// ---- DUTs/IO/PdoEntries/FSOE_BAA7477B.TcDUT
{attribute 'GeneratedUsingTerminal: EK1960-2600-0019'}
{attribute addProperty BoxType "EK1960-2600-0019"}
{attribute addProperty Id "FSoE_CommandUSINT1FSOUT_Module_1_Module_FaultBOOL1FSOUT_Module_2_Module_FaultBOOL1FSOUT_Module_3_Module_FaultBOOL1FSOUT_Module_4_Module_FaultBOOL1FSOUT_Module_5_Module_FaultBOOL1FSOUT_Module_6_Module_FaultBOOL1FSOUT_Relais_Module_Module_FaultBOOL1FSIN_Module_1_Channel_1_InputBOOL1FSIN_Module_1_Channel_2_InputBOOL1FSIN_Module_1_Module_FaultBOOL1FSIN_Module_2_Channel_1_InputBOOL1FSIN_Module_2_Channel_2_InputBOOL1FSIN_Module_2_Module_FaultBOOL1FSIN_Module_3_Channel_1_InputBOOL1FSIN_Module_3_Channel_2_InputBOOL1FSIN_Module_3_Module_FaultBOOL1FSoE_CRC_000UINT2FSIN_Module_4_Channel_1_InputBOOL1FSIN_Module_4_Channel_2_InputBOOL1FSIN_Module_4_Module_FaultBOOL1FSIN_Module_5_Channel_1_InputBOOL1FSIN_Module_5_Channel_2_InputBOOL1FSIN_Module_5_Module_FaultBOOL1FSIN_Module_6_Channel_1_InputBOOL1FSIN_Module_6_Channel_2_InputBOOL1FSIN_Module_6_Module_FaultBOOL1FSIN_Module_7_Channel_1_InputBOOL1FSIN_Module_7_Channel_2_InputBOOL1FSIN_Module_7_Module_FaultBOOL1FSIN_Module_8_Channel_1_InputBOOL1FSIN_Module_8_Channel_2_InputBOOL1FSIN_Module_8_Module_FaultBOOL1FSIN_Module_9_Channel_1_InputBOOL1FSoE_CRC_001UINT2FSIN_Module_9_Channel_2_InputBOOL1FSIN_Module_9_Module_Fault_1BOOL1FSIN_Module_9_Module_Fault_2BOOL1FSIN_Module_10_Channel_1_InputBOOL1FSIN_Module_10_Channel_2_InputBOOL1FSIN_Module_10_Module_Fault_1BOOL1FSIN_Module_10_Module_Fault_2BOOL1FSoE_CRC_002UINT2FSoE_Connection_IDUINT2"}
{attribute addProperty CRC "3131524987"}
{attribute addProperty Size "48"}
TYPE FSOE_BAA7477B :
STRUCT
	{attribute addProperty Name "FSoE_Command"}
	FSoE_Command : USINT;
	{attribute addProperty Name "FSOUT_Module_1_Module_Fault"}
	FSOUT_Module_1_Module_Fault : BOOL;
	{attribute addProperty Name "FSOUT_Module_2_Module_Fault"}
	FSOUT_Module_2_Module_Fault : BOOL;
	{attribute addProperty Name "FSOUT_Module_3_Module_Fault"}
	FSOUT_Module_3_Module_Fault : BOOL;
	{attribute addProperty Name "FSOUT_Module_4_Module_Fault"}
	FSOUT_Module_4_Module_Fault : BOOL;
	{attribute addProperty Name "FSOUT_Module_5_Module_Fault"}
	FSOUT_Module_5_Module_Fault : BOOL;
	{attribute addProperty Name "FSOUT_Module_6_Module_Fault"}
	FSOUT_Module_6_Module_Fault : BOOL;
	{attribute addProperty Name "FSOUT_Relais_Module_Module_Fault"}
	FSOUT_Relais_Module_Module_Fault : BOOL;
	{attribute addProperty Name "FSIN_Module_1_Channel_1_Input"}
	FSIN_Module_1_Channel_1_Input : BOOL;
	{attribute addProperty Name "FSIN_Module_1_Channel_2_Input"}
	FSIN_Module_1_Channel_2_Input : BOOL;
	{attribute addProperty Name "FSIN_Module_1_Module_Fault"}
	FSIN_Module_1_Module_Fault : BOOL;
	{attribute addProperty Name "FSIN_Module_2_Channel_1_Input"}
	FSIN_Module_2_Channel_1_Input : BOOL;
	{attribute addProperty Name "FSIN_Module_2_Channel_2_Input"}
	FSIN_Module_2_Channel_2_Input : BOOL;
	{attribute addProperty Name "FSIN_Module_2_Module_Fault"}
	FSIN_Module_2_Module_Fault : BOOL;
	{attribute addProperty Name "FSIN_Module_3_Channel_1_Input"}
	FSIN_Module_3_Channel_1_Input : BOOL;
	{attribute addProperty Name "FSIN_Module_3_Channel_2_Input"}
	FSIN_Module_3_Channel_2_Input : BOOL;
	{attribute addProperty Name "FSIN_Module_3_Module_Fault"}
	FSIN_Module_3_Module_Fault : BOOL;
	{attribute addProperty Name "FSoE_CRC_000"}
	FSoE_CRC_000 : UINT;
	{attribute addProperty Name "FSIN_Module_4_Channel_1_Input"}
	FSIN_Module_4_Channel_1_Input : BOOL;
	{attribute addProperty Name "FSIN_Module_4_Channel_2_Input"}
	FSIN_Module_4_Channel_2_Input : BOOL;
	{attribute addProperty Name "FSIN_Module_4_Module_Fault"}
	FSIN_Module_4_Module_Fault : BOOL;
	{attribute addProperty Name "FSIN_Module_5_Channel_1_Input"}
	FSIN_Module_5_Channel_1_Input : BOOL;
	{attribute addProperty Name "FSIN_Module_5_Channel_2_Input"}
	FSIN_Module_5_Channel_2_Input : BOOL;
	{attribute addProperty Name "FSIN_Module_5_Module_Fault"}
	FSIN_Module_5_Module_Fault : BOOL;
	{attribute addProperty Name "FSIN_Module_6_Channel_1_Input"}
	FSIN_Module_6_Channel_1_Input : BOOL;
	{attribute addProperty Name "FSIN_Module_6_Channel_2_Input"}
	FSIN_Module_6_Channel_2_Input : BOOL;
	{attribute addProperty Name "FSIN_Module_6_Module_Fault"}
	FSIN_Module_6_Module_Fault : BOOL;
	{attribute addProperty Name "FSIN_Module_7_Channel_1_Input"}
	FSIN_Module_7_Channel_1_Input : BOOL;
	{attribute addProperty Name "FSIN_Module_7_Channel_2_Input"}
	FSIN_Module_7_Channel_2_Input : BOOL;
	{attribute addProperty Name "FSIN_Module_7_Module_Fault"}
	FSIN_Module_7_Module_Fault : BOOL;
	{attribute addProperty Name "FSIN_Module_8_Channel_1_Input"}
	FSIN_Module_8_Channel_1_Input : BOOL;
	{attribute addProperty Name "FSIN_Module_8_Channel_2_Input"}
	FSIN_Module_8_Channel_2_Input : BOOL;
	{attribute addProperty Name "FSIN_Module_8_Module_Fault"}
	FSIN_Module_8_Module_Fault : BOOL;
	{attribute addProperty Name "FSIN_Module_9_Channel_1_Input"}
	FSIN_Module_9_Channel_1_Input : BOOL;
	{attribute addProperty Name "FSoE_CRC_001"}
	FSoE_CRC_001 : UINT;
	{attribute addProperty Name "FSIN_Module_9_Channel_2_Input"}
	FSIN_Module_9_Channel_2_Input : BOOL;
	{attribute addProperty Name "FSIN_Module_9_Module_Fault_1"}
	FSIN_Module_9_Module_Fault_1 : BOOL;
	{attribute addProperty Name "FSIN_Module_9_Module_Fault_2"}
	FSIN_Module_9_Module_Fault_2 : BOOL;
	{attribute addProperty Name "FSIN_Module_10_Channel_1_Input"}
	FSIN_Module_10_Channel_1_Input : BOOL;
	{attribute addProperty Name "FSIN_Module_10_Channel_2_Input"}
	FSIN_Module_10_Channel_2_Input : BOOL;
	{attribute addProperty Name "FSIN_Module_10_Module_Fault_1"}
	FSIN_Module_10_Module_Fault_1 : BOOL;
	{attribute addProperty Name "FSIN_Module_10_Module_Fault_2"}
	FSIN_Module_10_Module_Fault_2 : BOOL;
	{attribute addProperty Name "FSoE_CRC_002"}
	FSoE_CRC_002 : UINT;
	{attribute addProperty Name "FSoE_Connection_ID"}
	FSoE_Connection_ID : UINT;
END_STRUCT
END_TYPE

// ---- DUTs/IO/PdoEntries/FSOE_CEFF8C56.TcDUT
{attribute 'GeneratedUsingTerminal: EK1960-2600-0019'}
{attribute addProperty BoxType "EK1960-2600-0019"}
{attribute addProperty Id "FSoE_CommandUSINT1FSOUT_Module_1_Channel_1_OutputBOOL1FSOUT_Module_1_Channel_2_OutputBOOL1FSOUT_Module_1_Channel_3_OutputBOOL1FSOUT_Module_1_Channel_4_OutputBOOL1FSOUT_Module_1_ErrAckBOOL1FSOUT_Module_2_Channel_1_OutputBOOL1FSOUT_Module_2_Channel_2_OutputBOOL1FSOUT_Module_2_Channel_3_OutputBOOL1FSOUT_Module_2_Channel_4_OutputBOOL1FSOUT_Module_2_ErrAckBOOL1FSOUT_Module_3_Channel_1_OutputBOOL1FSOUT_Module_3_Channel_2_OutputBOOL1FSOUT_Module_3_Channel_3_OutputBOOL1FSOUT_Module_3_Channel_4_OutputBOOL1FSOUT_Module_3_ErrAckBOOL1FSOUT_Module_4_Channel_1_OutputBOOL1FSoE_CRC_000UINT2FSOUT_Module_4_Channel_2_OutputBOOL1FSOUT_Module_4_Channel_3_OutputBOOL1FSOUT_Module_4_Channel_4_OutputBOOL1FSOUT_Module_4_ErrAckBOOL1FSOUT_Module_5_Channel_1_OutputBOOL1FSOUT_Module_5_Channel_2_OutputBOOL1FSOUT_Module_5_Channel_3_OutputBOOL1FSOUT_Module_5_Channel_4_OutputBOOL1FSOUT_Module_5_ErrAckBOOL1FSOUT_Module_6_Channel_1_OutputBOOL1FSOUT_Module_6_Channel_2_OutputBOOL1FSOUT_Module_6_Channel_3_OutputBOOL1FSOUT_Module_6_Channel_4_OutputBOOL1FSOUT_Module_6_ErrAckBOOL1FSOUT_Relais_Module_Channel_1_OutputBOOL1FSOUT_Relais_Module_Channel_2_OutputBOOL1FSoE_CRC_001UINT2FSOUT_Relais_Module_Channel_3_OutputBOOL1FSOUT_Relais_Module_Channel_4_OutputBOOL1FSOUT_Relais_Module_ErrAckBOOL1FSIN_Module_1_ErrAckBOOL1FSIN_Module_2_ErrAckBOOL1FSIN_Module_3_ErrAckBOOL1FSIN_Module_4_ErrAckBOOL1FSIN_Module_5_ErrAckBOOL1FSIN_Module_6_ErrAckBOOL1FSIN_Module_7_ErrAckBOOL1FSIN_Module_8_ErrAckBOOL1FSIN_Module_9_ErrAck_1BOOL1FSIN_Module_9_ErrAck_2BOOL1FSIN_Module_10_ErrAck_1BOOL1FSIN_Module_10_ErrAck_2BOOL1FSoE_CRC_002UINT2FSoE_Connection_IDUINT2"}
{attribute addProperty CRC "3472854102"}
{attribute addProperty Size "56"}
TYPE FSOE_CEFF8C56 :
STRUCT
	{attribute addProperty Name "FSoE_Command"}
	FSoE_Command : USINT;
	{attribute addProperty Name "FSOUT_Module_1_Channel_1_Output"}
	FSOUT_Module_1_Channel_1_Output : BOOL;
	{attribute addProperty Name "FSOUT_Module_1_Channel_2_Output"}
	FSOUT_Module_1_Channel_2_Output : BOOL;
	{attribute addProperty Name "FSOUT_Module_1_Channel_3_Output"}
	FSOUT_Module_1_Channel_3_Output : BOOL;
	{attribute addProperty Name "FSOUT_Module_1_Channel_4_Output"}
	FSOUT_Module_1_Channel_4_Output : BOOL;
	{attribute addProperty Name "FSOUT_Module_1_ErrAck"}
	FSOUT_Module_1_ErrAck : BOOL;
	{attribute addProperty Name "FSOUT_Module_2_Channel_1_Output"}
	FSOUT_Module_2_Channel_1_Output : BOOL;
	{attribute addProperty Name "FSOUT_Module_2_Channel_2_Output"}
	FSOUT_Module_2_Channel_2_Output : BOOL;
	{attribute addProperty Name "FSOUT_Module_2_Channel_3_Output"}
	FSOUT_Module_2_Channel_3_Output : BOOL;
	{attribute addProperty Name "FSOUT_Module_2_Channel_4_Output"}
	FSOUT_Module_2_Channel_4_Output : BOOL;
	{attribute addProperty Name "FSOUT_Module_2_ErrAck"}
	FSOUT_Module_2_ErrAck : BOOL;
	{attribute addProperty Name "FSOUT_Module_3_Channel_1_Output"}
	FSOUT_Module_3_Channel_1_Output : BOOL;
	{attribute addProperty Name "FSOUT_Module_3_Channel_2_Output"}
	FSOUT_Module_3_Channel_2_Output : BOOL;
	{attribute addProperty Name "FSOUT_Module_3_Channel_3_Output"}
	FSOUT_Module_3_Channel_3_Output : BOOL;
	{attribute addProperty Name "FSOUT_Module_3_Channel_4_Output"}
	FSOUT_Module_3_Channel_4_Output : BOOL;
	{attribute addProperty Name "FSOUT_Module_3_ErrAck"}
	FSOUT_Module_3_ErrAck : BOOL;
	{attribute addProperty Name "FSOUT_Module_4_Channel_1_Output"}
	FSOUT_Module_4_Channel_1_Output : BOOL;
	{attribute addProperty Name "FSoE_CRC_000"}
	FSoE_CRC_000 : UINT;
	{attribute addProperty Name "FSOUT_Module_4_Channel_2_Output"}
	FSOUT_Module_4_Channel_2_Output : BOOL;
	{attribute addProperty Name "FSOUT_Module_4_Channel_3_Output"}
	FSOUT_Module_4_Channel_3_Output : BOOL;
	{attribute addProperty Name "FSOUT_Module_4_Channel_4_Output"}
	FSOUT_Module_4_Channel_4_Output : BOOL;
	{attribute addProperty Name "FSOUT_Module_4_ErrAck"}
	FSOUT_Module_4_ErrAck : BOOL;
	{attribute addProperty Name "FSOUT_Module_5_Channel_1_Output"}
	FSOUT_Module_5_Channel_1_Output : BOOL;
	{attribute addProperty Name "FSOUT_Module_5_Channel_2_Output"}
	FSOUT_Module_5_Channel_2_Output : BOOL;
	{attribute addProperty Name "FSOUT_Module_5_Channel_3_Output"}
	FSOUT_Module_5_Channel_3_Output : BOOL;
	{attribute addProperty Name "FSOUT_Module_5_Channel_4_Output"}
	FSOUT_Module_5_Channel_4_Output : BOOL;
	{attribute addProperty Name "FSOUT_Module_5_ErrAck"}
	FSOUT_Module_5_ErrAck : BOOL;
	{attribute addProperty Name "FSOUT_Module_6_Channel_1_Output"}
	FSOUT_Module_6_Channel_1_Output : BOOL;
	{attribute addProperty Name "FSOUT_Module_6_Channel_2_Output"}
	FSOUT_Module_6_Channel_2_Output : BOOL;
	{attribute addProperty Name "FSOUT_Module_6_Channel_3_Output"}
	FSOUT_Module_6_Channel_3_Output : BOOL;
	{attribute addProperty Name "FSOUT_Module_6_Channel_4_Output"}
	FSOUT_Module_6_Channel_4_Output : BOOL;
	{attribute addProperty Name "FSOUT_Module_6_ErrAck"}
	FSOUT_Module_6_ErrAck : BOOL;
	{attribute addProperty Name "FSOUT_Relais_Module_Channel_1_Output"}
	FSOUT_Relais_Module_Channel_1_Output : BOOL;
	{attribute addProperty Name "FSOUT_Relais_Module_Channel_2_Output"}
	FSOUT_Relais_Module_Channel_2_Output : BOOL;
	{attribute addProperty Name "FSoE_CRC_001"}
	FSoE_CRC_001 : UINT;
	{attribute addProperty Name "FSOUT_Relais_Module_Channel_3_Output"}
	FSOUT_Relais_Module_Channel_3_Output : BOOL;
	{attribute addProperty Name "FSOUT_Relais_Module_Channel_4_Output"}
	FSOUT_Relais_Module_Channel_4_Output : BOOL;
	{attribute addProperty Name "FSOUT_Relais_Module_ErrAck"}
	FSOUT_Relais_Module_ErrAck : BOOL;
	{attribute addProperty Name "FSIN_Module_1_ErrAck"}
	FSIN_Module_1_ErrAck : BOOL;
	{attribute addProperty Name "FSIN_Module_2_ErrAck"}
	FSIN_Module_2_ErrAck : BOOL;
	{attribute addProperty Name "FSIN_Module_3_ErrAck"}
	FSIN_Module_3_ErrAck : BOOL;
	{attribute addProperty Name "FSIN_Module_4_ErrAck"}
	FSIN_Module_4_ErrAck : BOOL;
	{attribute addProperty Name "FSIN_Module_5_ErrAck"}
	FSIN_Module_5_ErrAck : BOOL;
	{attribute addProperty Name "FSIN_Module_6_ErrAck"}
	FSIN_Module_6_ErrAck : BOOL;
	{attribute addProperty Name "FSIN_Module_7_ErrAck"}
	FSIN_Module_7_ErrAck : BOOL;
	{attribute addProperty Name "FSIN_Module_8_ErrAck"}
	FSIN_Module_8_ErrAck : BOOL;
	{attribute addProperty Name "FSIN_Module_9_ErrAck_1"}
	FSIN_Module_9_ErrAck_1 : BOOL;
	{attribute addProperty Name "FSIN_Module_9_ErrAck_2"}
	FSIN_Module_9_ErrAck_2 : BOOL;
	{attribute addProperty Name "FSIN_Module_10_ErrAck_1"}
	FSIN_Module_10_ErrAck_1 : BOOL;
	{attribute addProperty Name "FSIN_Module_10_ErrAck_2"}
	FSIN_Module_10_ErrAck_2 : BOOL;
	{attribute addProperty Name "FSoE_CRC_002"}
	FSoE_CRC_002 : UINT;
	{attribute addProperty Name "FSoE_Connection_ID"}
	FSoE_Connection_ID : UINT;
END_STRUCT
END_TYPE

// ---- DUTs/IO/PdoEntries/FSOE_E251F244.TcDUT
{attribute 'GeneratedUsingTerminal: EK1960-2600-0021'}
{attribute addProperty BoxType "EK1960-2600-0021"}
{attribute addProperty Id "FSoE_CommandUSINT1FSOUT_Module_1_Module_FaultBOOL1FSOUT_Module_2_Module_FaultBOOL1FSOUT_Module_3_Module_FaultBOOL1FSOUT_Module_4_Module_FaultBOOL1FSOUT_Module_5_Module_FaultBOOL1FSOUT_Module_6_Module_FaultBOOL1FSOUT_Relais_Module_Module_FaultBOOL1FSIN_Module_1_Channel_1_Input_X6_1BOOL1FSIN_Module_1_Channel_2_Input_X6_2BOOL1FSIN_Module_1_Module_FaultBOOL1FSIN_Module_2_Channel_1_Input_X6_3BOOL1FSIN_Module_2_Channel_2_Input_X6_4BOOL1FSIN_Module_2_Module_FaultBOOL1FSIN_Module_3_Channel_1_Input_X6_5BOOL1FSIN_Module_3_Channel_2_Input_X6_6BOOL1FSIN_Module_3_Module_FaultBOOL1FSoE_CRC_000UINT2FSIN_Module_4_Channel_1_Input_X6_7BOOL1FSIN_Module_4_Channel_2_Input_X6_8BOOL1FSIN_Module_4_Module_FaultBOOL1FSIN_Module_5_Channel_1_Input_X6_9BOOL1FSIN_Module_5_Channel_2_Input_X6_10BOOL1FSIN_Module_5_Module_FaultBOOL1FSIN_Module_6_Channel_1_Input_X8_1BOOL1FSIN_Module_6_Channel_2_Input_X8_2BOOL1FSIN_Module_6_Module_FaultBOOL1FSIN_Module_7_Channel_1_Input_X8_3BOOL1FSIN_Module_7_Channel_2_Input_X8_4BOOL1FSIN_Module_7_Module_FaultBOOL1FSIN_Module_8_Channel_1_Input_X8_5BOOL1FSIN_Module_8_Channel_2_Input_X8_6BOOL1FSIN_Module_8_Module_FaultBOOL1FSIN_Module_9_Channel_1_Input_X8_7BOOL1FSoE_CRC_001UINT2FSIN_Module_9_Channel_2_Input_X8_8BOOL1FSIN_Module_9_Module_Fault_1BOOL1FSIN_Module_9_Module_Fault_2BOOL1FSIN_Module_10_Channel_1_Input_X8_9BOOL1FSIN_Module_10_Channel_2_Input_X8_10BOOL1FSIN_Module_10_Module_Fault_1BOOL1FSIN_Module_10_Module_Fault_2BOOL1FSoE_CRC_002UINT2FSoE_Connection_IDUINT2"}
{attribute addProperty CRC "3797021252"}
{attribute addProperty Size "48"}
TYPE FSOE_E251F244 :
STRUCT
	{attribute addProperty Name "FSoE_Command"}
	FSoE_Command : USINT;
	{attribute addProperty Name "FSOUT_Module_1_Module_Fault"}
	FSOUT_Module_1_Module_Fault : BOOL;
	{attribute addProperty Name "FSOUT_Module_2_Module_Fault"}
	FSOUT_Module_2_Module_Fault : BOOL;
	{attribute addProperty Name "FSOUT_Module_3_Module_Fault"}
	FSOUT_Module_3_Module_Fault : BOOL;
	{attribute addProperty Name "FSOUT_Module_4_Module_Fault"}
	FSOUT_Module_4_Module_Fault : BOOL;
	{attribute addProperty Name "FSOUT_Module_5_Module_Fault"}
	FSOUT_Module_5_Module_Fault : BOOL;
	{attribute addProperty Name "FSOUT_Module_6_Module_Fault"}
	FSOUT_Module_6_Module_Fault : BOOL;
	{attribute addProperty Name "FSOUT_Relais_Module_Module_Fault"}
	FSOUT_Relais_Module_Module_Fault : BOOL;
	{attribute addProperty Name "FSIN_Module_1_Channel_1_Input_X6_1"}
	FSIN_Module_1_Channel_1_Input_X6_1 : BOOL;
	{attribute addProperty Name "FSIN_Module_1_Channel_2_Input_X6_2"}
	FSIN_Module_1_Channel_2_Input_X6_2 : BOOL;
	{attribute addProperty Name "FSIN_Module_1_Module_Fault"}
	FSIN_Module_1_Module_Fault : BOOL;
	{attribute addProperty Name "FSIN_Module_2_Channel_1_Input_X6_3"}
	FSIN_Module_2_Channel_1_Input_X6_3 : BOOL;
	{attribute addProperty Name "FSIN_Module_2_Channel_2_Input_X6_4"}
	FSIN_Module_2_Channel_2_Input_X6_4 : BOOL;
	{attribute addProperty Name "FSIN_Module_2_Module_Fault"}
	FSIN_Module_2_Module_Fault : BOOL;
	{attribute addProperty Name "FSIN_Module_3_Channel_1_Input_X6_5"}
	FSIN_Module_3_Channel_1_Input_X6_5 : BOOL;
	{attribute addProperty Name "FSIN_Module_3_Channel_2_Input_X6_6"}
	FSIN_Module_3_Channel_2_Input_X6_6 : BOOL;
	{attribute addProperty Name "FSIN_Module_3_Module_Fault"}
	FSIN_Module_3_Module_Fault : BOOL;
	{attribute addProperty Name "FSoE_CRC_000"}
	FSoE_CRC_000 : UINT;
	{attribute addProperty Name "FSIN_Module_4_Channel_1_Input_X6_7"}
	FSIN_Module_4_Channel_1_Input_X6_7 : BOOL;
	{attribute addProperty Name "FSIN_Module_4_Channel_2_Input_X6_8"}
	FSIN_Module_4_Channel_2_Input_X6_8 : BOOL;
	{attribute addProperty Name "FSIN_Module_4_Module_Fault"}
	FSIN_Module_4_Module_Fault : BOOL;
	{attribute addProperty Name "FSIN_Module_5_Channel_1_Input_X6_9"}
	FSIN_Module_5_Channel_1_Input_X6_9 : BOOL;
	{attribute addProperty Name "FSIN_Module_5_Channel_2_Input_X6_10"}
	FSIN_Module_5_Channel_2_Input_X6_10 : BOOL;
	{attribute addProperty Name "FSIN_Module_5_Module_Fault"}
	FSIN_Module_5_Module_Fault : BOOL;
	{attribute addProperty Name "FSIN_Module_6_Channel_1_Input_X8_1"}
	FSIN_Module_6_Channel_1_Input_X8_1 : BOOL;
	{attribute addProperty Name "FSIN_Module_6_Channel_2_Input_X8_2"}
	FSIN_Module_6_Channel_2_Input_X8_2 : BOOL;
	{attribute addProperty Name "FSIN_Module_6_Module_Fault"}
	FSIN_Module_6_Module_Fault : BOOL;
	{attribute addProperty Name "FSIN_Module_7_Channel_1_Input_X8_3"}
	FSIN_Module_7_Channel_1_Input_X8_3 : BOOL;
	{attribute addProperty Name "FSIN_Module_7_Channel_2_Input_X8_4"}
	FSIN_Module_7_Channel_2_Input_X8_4 : BOOL;
	{attribute addProperty Name "FSIN_Module_7_Module_Fault"}
	FSIN_Module_7_Module_Fault : BOOL;
	{attribute addProperty Name "FSIN_Module_8_Channel_1_Input_X8_5"}
	FSIN_Module_8_Channel_1_Input_X8_5 : BOOL;
	{attribute addProperty Name "FSIN_Module_8_Channel_2_Input_X8_6"}
	FSIN_Module_8_Channel_2_Input_X8_6 : BOOL;
	{attribute addProperty Name "FSIN_Module_8_Module_Fault"}
	FSIN_Module_8_Module_Fault : BOOL;
	{attribute addProperty Name "FSIN_Module_9_Channel_1_Input_X8_7"}
	FSIN_Module_9_Channel_1_Input_X8_7 : BOOL;
	{attribute addProperty Name "FSoE_CRC_001"}
	FSoE_CRC_001 : UINT;
	{attribute addProperty Name "FSIN_Module_9_Channel_2_Input_X8_8"}
	FSIN_Module_9_Channel_2_Input_X8_8 : BOOL;
	{attribute addProperty Name "FSIN_Module_9_Module_Fault_1"}
	FSIN_Module_9_Module_Fault_1 : BOOL;
	{attribute addProperty Name "FSIN_Module_9_Module_Fault_2"}
	FSIN_Module_9_Module_Fault_2 : BOOL;
	{attribute addProperty Name "FSIN_Module_10_Channel_1_Input_X8_9"}
	FSIN_Module_10_Channel_1_Input_X8_9 : BOOL;
	{attribute addProperty Name "FSIN_Module_10_Channel_2_Input_X8_10"}
	FSIN_Module_10_Channel_2_Input_X8_10 : BOOL;
	{attribute addProperty Name "FSIN_Module_10_Module_Fault_1"}
	FSIN_Module_10_Module_Fault_1 : BOOL;
	{attribute addProperty Name "FSIN_Module_10_Module_Fault_2"}
	FSIN_Module_10_Module_Fault_2 : BOOL;
	{attribute addProperty Name "FSoE_CRC_002"}
	FSoE_CRC_002 : UINT;
	{attribute addProperty Name "FSoE_Connection_ID"}
	FSoE_Connection_ID : UINT;
END_STRUCT
END_TYPE

// ---- DUTs/IO/PdoEntries/FSOE_CDFABDDF.TcDUT
{attribute 'GeneratedUsingTerminal: EK1960-2600-0021'}
{attribute addProperty BoxType "EK1960-2600-0021"}
{attribute addProperty Id "FSoE_CommandUSINT1FSOUT_Module_1_Channel_1_Output_X5_1BOOL1FSOUT_Module_1_Channel_2_Output_X5_2BOOL1FSOUT_Module_1_Channel_3_Output_X5_3BOOL1FSOUT_Module_1_Channel_4_Output_X5_4BOOL1FSOUT_Module_1_ErrAckBOOL1FSOUT_Module_2_Channel_1_Output_X5_5BOOL1FSOUT_Module_2_Channel_2_Output_X5_6BOOL1FSOUT_Module_2_Channel_3_Output_X5_7BOOL1FSOUT_Module_2_Channel_4_Output_X5_8BOOL1FSOUT_Module_2_ErrAckBOOL1FSOUT_Module_3_Channel_1_Output_X7_1BOOL1FSOUT_Module_3_Channel_2_Output_X7_2BOOL1FSOUT_Module_3_Channel_3_Output_X7_3BOOL1FSOUT_Module_3_Channel_4_Output_X7_4BOOL1FSOUT_Module_3_ErrAckBOOL1FSOUT_Module_4_Channel_1_Output_X7_5BOOL1FSoE_CRC_000UINT2FSOUT_Module_4_Channel_2_Output_X7_6BOOL1FSOUT_Module_4_Channel_3_Output_X7_7BOOL1FSOUT_Module_4_Channel_4_Output_X7_8BOOL1FSOUT_Module_4_ErrAckBOOL1FSOUT_Module_5_Channel_1_Output_X9_1BOOL1FSOUT_Module_5_Channel_2_Output_X9_2BOOL1FSOUT_Module_5_Channel_3_Output_X9_3BOOL1FSOUT_Module_5_Channel_4_Output_X9_4BOOL1FSOUT_Module_5_ErrAckBOOL1FSOUT_Module_6_Channel_1_Output_X9_5BOOL1FSOUT_Module_6_Channel_2_Output_X9_6BOOL1FSOUT_Module_6_Channel_3_Output_X9_7BOOL1FSOUT_Module_6_Channel_4_Output_X9_8BOOL1FSOUT_Module_6_ErrAckBOOL1FSOUT_Relais_Module_Channel_1_Output_X4_1_X4_5BOOL1FSOUT_Relais_Module_Channel_2_Output_X4_2_X4_6BOOL1FSoE_CRC_001UINT2FSOUT_Relais_Module_Channel_3_Output_X4_3_X4_7BOOL1FSOUT_Relais_Module_Channel_4_Output_X4_4_X4_8BOOL1FSOUT_Relais_Module_ErrAckBOOL1FSIN_Module_1_ErrAckBOOL1FSIN_Module_2_ErrAckBOOL1FSIN_Module_3_ErrAckBOOL1FSIN_Module_4_ErrAckBOOL1FSIN_Module_5_ErrAckBOOL1FSIN_Module_6_ErrAckBOOL1FSIN_Module_7_ErrAckBOOL1FSIN_Module_8_ErrAckBOOL1FSIN_Module_9_Err_Ack_1BOOL1FSIN_Module_9_Err_Ack_2BOOL1FSIN_Module_10_Err_Ack_1BOOL1FSIN_Module_10_Err_Ack_2BOOL1FSoE_CRC_002UINT2FSoE_Connection_IDUINT2"}
{attribute addProperty CRC "3455761887"}
{attribute addProperty Size "56"}
TYPE FSOE_CDFABDDF :
STRUCT
	{attribute addProperty Name "FSoE_Command"}
	FSoE_Command : USINT;
	{attribute addProperty Name "FSOUT_Module_1_Channel_1_Output_X5_1"}
	FSOUT_Module_1_Channel_1_Output_X5_1 : BOOL;
	{attribute addProperty Name "FSOUT_Module_1_Channel_2_Output_X5_2"}
	FSOUT_Module_1_Channel_2_Output_X5_2 : BOOL;
	{attribute addProperty Name "FSOUT_Module_1_Channel_3_Output_X5_3"}
	FSOUT_Module_1_Channel_3_Output_X5_3 : BOOL;
	{attribute addProperty Name "FSOUT_Module_1_Channel_4_Output_X5_4"}
	FSOUT_Module_1_Channel_4_Output_X5_4 : BOOL;
	{attribute addProperty Name "FSOUT_Module_1_ErrAck"}
	FSOUT_Module_1_ErrAck : BOOL;
	{attribute addProperty Name "FSOUT_Module_2_Channel_1_Output_X5_5"}
	FSOUT_Module_2_Channel_1_Output_X5_5 : BOOL;
	{attribute addProperty Name "FSOUT_Module_2_Channel_2_Output_X5_6"}
	FSOUT_Module_2_Channel_2_Output_X5_6 : BOOL;
	{attribute addProperty Name "FSOUT_Module_2_Channel_3_Output_X5_7"}
	FSOUT_Module_2_Channel_3_Output_X5_7 : BOOL;
	{attribute addProperty Name "FSOUT_Module_2_Channel_4_Output_X5_8"}
	FSOUT_Module_2_Channel_4_Output_X5_8 : BOOL;
	{attribute addProperty Name "FSOUT_Module_2_ErrAck"}
	FSOUT_Module_2_ErrAck : BOOL;
	{attribute addProperty Name "FSOUT_Module_3_Channel_1_Output_X7_1"}
	FSOUT_Module_3_Channel_1_Output_X7_1 : BOOL;
	{attribute addProperty Name "FSOUT_Module_3_Channel_2_Output_X7_2"}
	FSOUT_Module_3_Channel_2_Output_X7_2 : BOOL;
	{attribute addProperty Name "FSOUT_Module_3_Channel_3_Output_X7_3"}
	FSOUT_Module_3_Channel_3_Output_X7_3 : BOOL;
	{attribute addProperty Name "FSOUT_Module_3_Channel_4_Output_X7_4"}
	FSOUT_Module_3_Channel_4_Output_X7_4 : BOOL;
	{attribute addProperty Name "FSOUT_Module_3_ErrAck"}
	FSOUT_Module_3_ErrAck : BOOL;
	{attribute addProperty Name "FSOUT_Module_4_Channel_1_Output_X7_5"}
	FSOUT_Module_4_Channel_1_Output_X7_5 : BOOL;
	{attribute addProperty Name "FSoE_CRC_000"}
	FSoE_CRC_000 : UINT;
	{attribute addProperty Name "FSOUT_Module_4_Channel_2_Output_X7_6"}
	FSOUT_Module_4_Channel_2_Output_X7_6 : BOOL;
	{attribute addProperty Name "FSOUT_Module_4_Channel_3_Output_X7_7"}
	FSOUT_Module_4_Channel_3_Output_X7_7 : BOOL;
	{attribute addProperty Name "FSOUT_Module_4_Channel_4_Output_X7_8"}
	FSOUT_Module_4_Channel_4_Output_X7_8 : BOOL;
	{attribute addProperty Name "FSOUT_Module_4_ErrAck"}
	FSOUT_Module_4_ErrAck : BOOL;
	{attribute addProperty Name "FSOUT_Module_5_Channel_1_Output_X9_1"}
	FSOUT_Module_5_Channel_1_Output_X9_1 : BOOL;
	{attribute addProperty Name "FSOUT_Module_5_Channel_2_Output_X9_2"}
	FSOUT_Module_5_Channel_2_Output_X9_2 : BOOL;
	{attribute addProperty Name "FSOUT_Module_5_Channel_3_Output_X9_3"}
	FSOUT_Module_5_Channel_3_Output_X9_3 : BOOL;
	{attribute addProperty Name "FSOUT_Module_5_Channel_4_Output_X9_4"}
	FSOUT_Module_5_Channel_4_Output_X9_4 : BOOL;
	{attribute addProperty Name "FSOUT_Module_5_ErrAck"}
	FSOUT_Module_5_ErrAck : BOOL;
	{attribute addProperty Name "FSOUT_Module_6_Channel_1_Output_X9_5"}
	FSOUT_Module_6_Channel_1_Output_X9_5 : BOOL;
	{attribute addProperty Name "FSOUT_Module_6_Channel_2_Output_X9_6"}
	FSOUT_Module_6_Channel_2_Output_X9_6 : BOOL;
	{attribute addProperty Name "FSOUT_Module_6_Channel_3_Output_X9_7"}
	FSOUT_Module_6_Channel_3_Output_X9_7 : BOOL;
	{attribute addProperty Name "FSOUT_Module_6_Channel_4_Output_X9_8"}
	FSOUT_Module_6_Channel_4_Output_X9_8 : BOOL;
	{attribute addProperty Name "FSOUT_Module_6_ErrAck"}
	FSOUT_Module_6_ErrAck : BOOL;
	{attribute addProperty Name "FSOUT_Relais_Module_Channel_1_Output_X4_1_X4_5"}
	FSOUT_Relais_Module_Channel_1_Output_X4_1_X4_5 : BOOL;
	{attribute addProperty Name "FSOUT_Relais_Module_Channel_2_Output_X4_2_X4_6"}
	FSOUT_Relais_Module_Channel_2_Output_X4_2_X4_6 : BOOL;
	{attribute addProperty Name "FSoE_CRC_001"}
	FSoE_CRC_001 : UINT;
	{attribute addProperty Name "FSOUT_Relais_Module_Channel_3_Output_X4_3_X4_7"}
	FSOUT_Relais_Module_Channel_3_Output_X4_3_X4_7 : BOOL;
	{attribute addProperty Name "FSOUT_Relais_Module_Channel_4_Output_X4_4_X4_8"}
	FSOUT_Relais_Module_Channel_4_Output_X4_4_X4_8 : BOOL;
	{attribute addProperty Name "FSOUT_Relais_Module_ErrAck"}
	FSOUT_Relais_Module_ErrAck : BOOL;
	{attribute addProperty Name "FSIN_Module_1_ErrAck"}
	FSIN_Module_1_ErrAck : BOOL;
	{attribute addProperty Name "FSIN_Module_2_ErrAck"}
	FSIN_Module_2_ErrAck : BOOL;
	{attribute addProperty Name "FSIN_Module_3_ErrAck"}
	FSIN_Module_3_ErrAck : BOOL;
	{attribute addProperty Name "FSIN_Module_4_ErrAck"}
	FSIN_Module_4_ErrAck : BOOL;
	{attribute addProperty Name "FSIN_Module_5_ErrAck"}
	FSIN_Module_5_ErrAck : BOOL;
	{attribute addProperty Name "FSIN_Module_6_ErrAck"}
	FSIN_Module_6_ErrAck : BOOL;
	{attribute addProperty Name "FSIN_Module_7_ErrAck"}
	FSIN_Module_7_ErrAck : BOOL;
	{attribute addProperty Name "FSIN_Module_8_ErrAck"}
	FSIN_Module_8_ErrAck : BOOL;
	{attribute addProperty Name "FSIN_Module_9_Err_Ack_1"}
	FSIN_Module_9_Err_Ack_1 : BOOL;
	{attribute addProperty Name "FSIN_Module_9_Err_Ack_2"}
	FSIN_Module_9_Err_Ack_2 : BOOL;
	{attribute addProperty Name "FSIN_Module_10_Err_Ack_1"}
	FSIN_Module_10_Err_Ack_1 : BOOL;
	{attribute addProperty Name "FSIN_Module_10_Err_Ack_2"}
	FSIN_Module_10_Err_Ack_2 : BOOL;
	{attribute addProperty Name "FSoE_CRC_002"}
	FSoE_CRC_002 : UINT;
	{attribute addProperty Name "FSoE_Connection_ID"}
	FSoE_Connection_ID : UINT;
END_STRUCT
END_TYPE

// ---- DUTs/IO/PDOs/InfoData_6F19DB2B.TcDUT
{attribute 'GeneratedUsingTerminal: EK1100-0000-0018'}
{attribute addProperty BoxType "EK1100-0000-0018"}
{attribute addProperty Id "StateAT %I*UINT2"}
{attribute addProperty CRC "1863965483"}
{attribute addProperty Size "2"}
TYPE InfoData_6F19DB2B :
STRUCT
	{attribute addProperty Name "State"}
	State AT %I* : UINT;
END_STRUCT
END_TYPE

// ---- DUTs/IO/PDOs/ID_07C9D28F.TcDUT
{attribute 'GeneratedUsingTerminal: EK1101-0000-0016'}
{attribute addProperty BoxType "EK1101-0000-0016"}
{attribute addProperty Id "IDAT %I*UINT2"}
{attribute addProperty CRC "130667151"}
{attribute addProperty Size "2"}
TYPE ID_07C9D28F EXTENDS InputBase_8311D824 :
STRUCT
	{attribute addProperty Name "ID"}
	ID AT %I* : UINT;
END_STRUCT
END_TYPE

// ---- DUTs/IO/PDOs/WcState_9091E0EB.TcDUT
{attribute 'GeneratedUsingTerminal: EK1101-0000-0016'}
{attribute addProperty BoxType "EK1101-0000-0016"}
{attribute addProperty Id "WcStateAT %I*BOOL1InputToggleAT %I*BOOL1"}
{attribute addProperty CRC "2425479403"}
{attribute addProperty Size "2"}
TYPE WcState_9091E0EB :
STRUCT
	{attribute addProperty Name "WcState"}
	WcState AT %I* : BOOL;
	{attribute addProperty Name "InputToggle"}
	InputToggle AT %I* : BOOL;
END_STRUCT
END_TYPE

// ---- DUTs/IO/PDOs/Status_Us_B1E819A2.TcDUT
{attribute 'GeneratedUsingTerminal: EK1300-0000-0017'}
{attribute addProperty BoxType "EK1300-0000-0017"}
{attribute addProperty Id "UndervoltageAT %I*BOOL1"}
{attribute addProperty CRC "2984778146"}
{attribute addProperty Size "1"}
TYPE Status_Us_B1E819A2 EXTENDS InputBase_8311D824 :
STRUCT
	{attribute addProperty Name "Undervoltage"}
	Undervoltage AT %I* : BOOL;
END_STRUCT
END_TYPE

// ---- DUTs/IO/PDOs/Status_Up_B1E819A2.TcDUT
{attribute 'GeneratedUsingTerminal: EK1300-0000-0017'}
{attribute addProperty BoxType "EK1300-0000-0017"}
{attribute addProperty Id "UndervoltageAT %I*BOOL1"}
{attribute addProperty CRC "2984778146"}
{attribute addProperty Size "1"}
TYPE Status_Up_B1E819A2 EXTENDS InputBase_8311D824 :
STRUCT
	{attribute addProperty Name "Undervoltage"}
	Undervoltage AT %I* : BOOL;
END_STRUCT
END_TYPE

// ---- DUTs/IO/PDOs/Channel_830843C1.TcDUT
{attribute 'GeneratedUsingTerminal: EK1814-0000-0016'}
{attribute addProperty BoxType "EK1814-0000-0016"}
{attribute addProperty Id "InputAT %I*BOOL1"}
{attribute addProperty CRC "2198356929"}
{attribute addProperty Size "1"}
TYPE Channel_830843C1 EXTENDS InputBase_8311D824 :
STRUCT
	{attribute addProperty Name "Input"}
	Input AT %I* : BOOL;
END_STRUCT
END_TYPE

// ---- DUTs/IO/PDOs/Channel_42CA91F7.TcDUT
{attribute 'GeneratedUsingTerminal: EK1814-0000-0016'}
{attribute addProperty BoxType "EK1814-0000-0016"}
{attribute addProperty Id "OutputAT %Q*BOOL1"}
{attribute addProperty CRC "1120571895"}
{attribute addProperty Size "1"}
TYPE Channel_42CA91F7 EXTENDS OutputBase_10CEE7DE :
STRUCT
	{attribute addProperty Name "Output"}
	Output AT %Q* : BOOL;
END_STRUCT
END_TYPE

// ---- DUTs/IO/PDOs/WcState_0B2B16F9.TcDUT
{attribute 'GeneratedUsingTerminal: EK1828-0010-0016'}
{attribute addProperty BoxType "EK1828-0010-0016"}
{attribute addProperty Id "WcStateAT %I*BOOL1"}
{attribute addProperty CRC "187373305"}
{attribute addProperty Size "1"}
TYPE WcState_0B2B16F9 :
STRUCT
	{attribute addProperty Name "WcState"}
	WcState AT %I* : BOOL;
END_STRUCT
END_TYPE

// ---- DUTs/IO/PDOs/MMS_Device_Inputs_ADC3123E.TcDUT
{attribute 'GeneratedUsingTerminal: EKM1101-0000-0016'}
{attribute addProperty BoxType "EKM1101-0000-0016"}
{attribute addProperty Id "StatusAT %I*Status_9847B4EF5"}
{attribute addProperty CRC "2915242558"}
{attribute addProperty Size "5"}
TYPE MMS_Device_Inputs_ADC3123E EXTENDS InputBase_8311D824 :
STRUCT
	{attribute addProperty Name "Status"}
	Status AT %I* : Status_9847B4EF;
END_STRUCT
END_TYPE

// ---- DUTs/IO/PDOs/MMS_Acceleration_Status_11769099.TcDUT
{attribute 'GeneratedUsingTerminal: EKM1101-0000-0016'}
{attribute addProperty BoxType "EKM1101-0000-0016"}
{attribute addProperty Id "StatusAT %I*Status_BA3D1C5D7Number_of_samplesAT %I*UINT2"}
{attribute addProperty CRC "292982937"}
{attribute addProperty Size "9"}
TYPE MMS_Acceleration_Status_11769099 EXTENDS InputBase_8311D824 :
STRUCT
	{attribute addProperty Name "Status"}
	Status AT %I* : Status_BA3D1C5D;
	{attribute addProperty Name "Number_of_samples"}
	Number_of_samples AT %I* : UINT;
END_STRUCT
END_TYPE

// ---- DUTs/IO/PDOs/MMS_Acceleration_X_Axis_80E77D6A.TcDUT
{attribute 'GeneratedUsingTerminal: EKM1101-0000-0016'}
{attribute addProperty BoxType "EKM1101-0000-0016"}
{attribute addProperty Id "ValueAT %I*INT2"}
{attribute addProperty CRC "2162654570"}
{attribute addProperty Size "2"}
TYPE MMS_Acceleration_X_Axis_80E77D6A EXTENDS InputBase_8311D824 :
STRUCT
	{attribute addProperty Name "Value"}
	Value AT %I* : INT;
END_STRUCT
END_TYPE

// ---- DUTs/IO/PDOs/MMS_Acceleration_Y_Axis_80E77D6A.TcDUT
{attribute 'GeneratedUsingTerminal: EKM1101-0000-0016'}
{attribute addProperty BoxType "EKM1101-0000-0016"}
{attribute addProperty Id "ValueAT %I*INT2"}
{attribute addProperty CRC "2162654570"}
{attribute addProperty Size "2"}
TYPE MMS_Acceleration_Y_Axis_80E77D6A EXTENDS InputBase_8311D824 :
STRUCT
	{attribute addProperty Name "Value"}
	Value AT %I* : INT;
END_STRUCT
END_TYPE

// ---- DUTs/IO/PDOs/MMS_Acceleration_Z_Axis_80E77D6A.TcDUT
{attribute 'GeneratedUsingTerminal: EKM1101-0000-0016'}
{attribute addProperty BoxType "EKM1101-0000-0016"}
{attribute addProperty Id "ValueAT %I*INT2"}
{attribute addProperty CRC "2162654570"}
{attribute addProperty Size "2"}
TYPE MMS_Acceleration_Z_Axis_80E77D6A EXTENDS InputBase_8311D824 :
STRUCT
	{attribute addProperty Name "Value"}
	Value AT %I* : INT;
END_STRUCT
END_TYPE

// ---- DUTs/IO/PDOs/MMS_Acceleration_Timestamp_8B9FE1A2.TcDUT
{attribute 'GeneratedUsingTerminal: EKM1101-0000-0016'}
{attribute addProperty BoxType "EKM1101-0000-0016"}
{attribute addProperty Id "TimestampAT %I*ULINT8"}
{attribute addProperty CRC "2342511010"}
{attribute addProperty Size "8"}
TYPE MMS_Acceleration_Timestamp_8B9FE1A2 EXTENDS InputBase_8311D824 :
STRUCT
	{attribute addProperty Name "Timestamp"}
	Timestamp AT %I* : ULINT;
END_STRUCT
END_TYPE

// ---- DUTs/IO/PDOs/MMS_Voltage_Us_In_Inputs_60D55C72.TcDUT
{attribute 'GeneratedUsingTerminal: EKM1101-0000-0016'}
{attribute addProperty BoxType "EKM1101-0000-0016"}
{attribute addProperty Id "StatusAT %I*Status_F2CE6D917ValueAT %I*REAL4"}
{attribute addProperty CRC "1624595570"}
{attribute addProperty Size "11"}
TYPE MMS_Voltage_Us_In_Inputs_60D55C72 EXTENDS InputBase_8311D824 :
STRUCT
	{attribute addProperty Name "Status"}
	Status AT %I* : Status_F2CE6D91;
	{attribute addProperty Name "Value"}
	Value AT %I* : REAL;
END_STRUCT
END_TYPE

// ---- DUTs/IO/PDOs/MMS_Voltage_Up_In_Inputs_60D55C72.TcDUT
{attribute 'GeneratedUsingTerminal: EKM1101-0000-0016'}
{attribute addProperty BoxType "EKM1101-0000-0016"}
{attribute addProperty Id "StatusAT %I*Status_F2CE6D917ValueAT %I*REAL4"}
{attribute addProperty CRC "1624595570"}
{attribute addProperty Size "11"}
TYPE MMS_Voltage_Up_In_Inputs_60D55C72 EXTENDS InputBase_8311D824 :
STRUCT
	{attribute addProperty Name "Status"}
	Status AT %I* : Status_F2CE6D91;
	{attribute addProperty Name "Value"}
	Value AT %I* : REAL;
END_STRUCT
END_TYPE

// ---- DUTs/IO/PDOs/MMS_Voltage_Up_Out_Inputs_60D55C72.TcDUT
{attribute 'GeneratedUsingTerminal: EKM1101-0000-0016'}
{attribute addProperty BoxType "EKM1101-0000-0016"}
{attribute addProperty Id "StatusAT %I*Status_F2CE6D917ValueAT %I*REAL4"}
{attribute addProperty CRC "1624595570"}
{attribute addProperty Size "11"}
TYPE MMS_Voltage_Up_Out_Inputs_60D55C72 EXTENDS InputBase_8311D824 :
STRUCT
	{attribute addProperty Name "Status"}
	Status AT %I* : Status_F2CE6D91;
	{attribute addProperty Name "Value"}
	Value AT %I* : REAL;
END_STRUCT
END_TYPE

// ---- DUTs/IO/PDOs/MMS_Device_Outputs_E6E6F9D1.TcDUT
{attribute 'GeneratedUsingTerminal: EKM1101-0000-0016'}
{attribute addProperty BoxType "EKM1101-0000-0016"}
{attribute addProperty Id "ControlAT %Q*Control_EBEDCF761"}
{attribute addProperty CRC "3873896913"}
{attribute addProperty Size "1"}
TYPE MMS_Device_Outputs_E6E6F9D1 EXTENDS OutputBase_10CEE7DE :
STRUCT
	{attribute addProperty Name "Control"}
	Control AT %Q* : Control_EBEDCF76;
END_STRUCT
END_TYPE

// ---- DUTs/IO/PDOs/InfoData_BEF6B88E.TcDUT
{attribute 'GeneratedUsingTerminal: EKM1101-0000-0016'}
{attribute addProperty BoxType "EKM1101-0000-0016"}
{attribute addProperty Id "AdsAddrAT %I*AMSADDR8DcOutputShiftAT %I*DINT4DcInputShiftAT %I*DINT4StateAT %I*UINT2"}
{attribute addProperty CRC "3203840142"}
{attribute addProperty Size "18"}
TYPE InfoData_BEF6B88E EXTENDS InputBase_8311D824 :
STRUCT
	{attribute addProperty Name "AdsAddr"}
	AdsAddr AT %I* : AMSADDR;
	{attribute addProperty Name "DcOutputShift"}
	DcOutputShift AT %I* : DINT;
	{attribute addProperty Name "DcInputShift"}
	DcInputShift AT %I* : DINT;
	{attribute addProperty Name "State"}
	State AT %I* : UINT;
END_STRUCT
END_TYPE

// ---- DUTs/IO/PDOs/FSoE_Inputs_9283FC69.TcDUT
{attribute 'GeneratedUsingTerminal: EK1960-0000-0019'}
{attribute addProperty BoxType "EK1960-0000-0019"}
{attribute addProperty Id "FSOEAT %I*FSOE_BBDEEE9E47"}
{attribute addProperty CRC "2458123369"}
{attribute addProperty Size "47"}
TYPE FSoE_Inputs_9283FC69 EXTENDS InputBase_8311D824 :
STRUCT
	{attribute addProperty Name "FSOE"}
	FSOE AT %I* : FSOE_BBDEEE9E;
END_STRUCT
END_TYPE

// ---- DUTs/IO/PDOs/FSoE_Outputs_79E75DAB.TcDUT
{attribute 'GeneratedUsingTerminal: EK1960-0000-0019'}
{attribute addProperty BoxType "EK1960-0000-0019"}
{attribute addProperty Id "FSOEAT %Q*FSOE_BAC7BF2151"}
{attribute addProperty CRC "2045205931"}
{attribute addProperty Size "51"}
TYPE FSoE_Outputs_79E75DAB EXTENDS OutputBase_10CEE7DE :
STRUCT
	{attribute addProperty Name "FSOE"}
	FSOE AT %Q* : FSOE_BAC7BF21;
END_STRUCT
END_TYPE

// ---- DUTs/IO/PDOs/Outputs_63C46CC8.TcDUT
{attribute 'GeneratedUsingTerminal: EK1960-0000-0019'}
{attribute addProperty BoxType "EK1960-0000-0019"}
{attribute addProperty Id "Module_1_Channel_1_Standard_Output_X5_1AT %Q*BOOL1Module_1_Channel_2_Standard_Output_X5_2AT %Q*BOOL1Module_1_Channel_3_Standard_Output_X5_3AT %Q*BOOL1Module_1_Channel_4_Standard_Output_X5_4AT %Q*BOOL1Module_2_Channel_1_Standard_Output_X5_5AT %Q*BOOL1Module_2_Channel_2_Standard_Output_X5_6AT %Q*BOOL1Module_2_Channel_3_Standard_Output_X5_7AT %Q*BOOL1Module_2_Channel_4_Standard_Output_X5_8AT %Q*BOOL1Module_3_Channel_1_Standard_Output_X7_1AT %Q*BOOL1Module_3_Channel_2_Standard_Output_X7_2AT %Q*BOOL1Module_3_Channel_3_Standard_Output_X7_3AT %Q*BOOL1Module_3_Channel_4_Standard_Output_X7_4AT %Q*BOOL1Module_4_Channel_1_Standard_Output_X7_5AT %Q*BOOL1Module_4_Channel_2_Standard_Output_X7_6AT %Q*BOOL1Module_4_Channel_3_Standard_Output_X7_7AT %Q*BOOL1Module_4_Channel_4_Standard_Output_X7_8AT %Q*BOOL1Module_5_Channel_1_Standard_Output_X9_1AT %Q*BOOL1Module_5_Channel_2_Standard_Output_X9_2AT %Q*BOOL1Module_5_Channel_3_Standard_Output_X9_3AT %Q*BOOL1Module_5_Channel_4_Standard_Output_X9_4AT %Q*BOOL1Module_6_Channel_1_Standard_Output_X9_5AT %Q*BOOL1Module_6_Channel_2_Standard_Output_X9_6AT %Q*BOOL1Module_6_Channel_3_Standard_Output_X9_7AT %Q*BOOL1Module_6_Channel_4_Standard_Output_X9_8AT %Q*BOOL1Relais_Module_Channel_1_Standard_Output_X4_1_X4_5AT %Q*BOOL1Relais_Module_Channel_2_Standard_Output_X4_2_X4_6AT %Q*BOOL1Relais_Module_Channel_3_Standard_Output_X4_3_X4_7AT %Q*BOOL1Relais_Module_Channel_4_Standard_Output_X4_4_X4_8AT %Q*BOOL1"}
{attribute addProperty CRC "1673817288"}
{attribute addProperty Size "28"}
TYPE Outputs_63C46CC8 EXTENDS OutputBase_10CEE7DE :
STRUCT
	{attribute addProperty Name "Module_1_Channel_1_Standard_Output_X5_1"}
	Module_1_Channel_1_Standard_Output_X5_1 AT %Q* : BOOL;
	{attribute addProperty Name "Module_1_Channel_2_Standard_Output_X5_2"}
	Module_1_Channel_2_Standard_Output_X5_2 AT %Q* : BOOL;
	{attribute addProperty Name "Module_1_Channel_3_Standard_Output_X5_3"}
	Module_1_Channel_3_Standard_Output_X5_3 AT %Q* : BOOL;
	{attribute addProperty Name "Module_1_Channel_4_Standard_Output_X5_4"}
	Module_1_Channel_4_Standard_Output_X5_4 AT %Q* : BOOL;
	{attribute addProperty Name "Module_2_Channel_1_Standard_Output_X5_5"}
	Module_2_Channel_1_Standard_Output_X5_5 AT %Q* : BOOL;
	{attribute addProperty Name "Module_2_Channel_2_Standard_Output_X5_6"}
	Module_2_Channel_2_Standard_Output_X5_6 AT %Q* : BOOL;
	{attribute addProperty Name "Module_2_Channel_3_Standard_Output_X5_7"}
	Module_2_Channel_3_Standard_Output_X5_7 AT %Q* : BOOL;
	{attribute addProperty Name "Module_2_Channel_4_Standard_Output_X5_8"}
	Module_2_Channel_4_Standard_Output_X5_8 AT %Q* : BOOL;
	{attribute addProperty Name "Module_3_Channel_1_Standard_Output_X7_1"}
	Module_3_Channel_1_Standard_Output_X7_1 AT %Q* : BOOL;
	{attribute addProperty Name "Module_3_Channel_2_Standard_Output_X7_2"}
	Module_3_Channel_2_Standard_Output_X7_2 AT %Q* : BOOL;
	{attribute addProperty Name "Module_3_Channel_3_Standard_Output_X7_3"}
	Module_3_Channel_3_Standard_Output_X7_3 AT %Q* : BOOL;
	{attribute addProperty Name "Module_3_Channel_4_Standard_Output_X7_4"}
	Module_3_Channel_4_Standard_Output_X7_4 AT %Q* : BOOL;
	{attribute addProperty Name "Module_4_Channel_1_Standard_Output_X7_5"}
	Module_4_Channel_1_Standard_Output_X7_5 AT %Q* : BOOL;
	{attribute addProperty Name "Module_4_Channel_2_Standard_Output_X7_6"}
	Module_4_Channel_2_Standard_Output_X7_6 AT %Q* : BOOL;
	{attribute addProperty Name "Module_4_Channel_3_Standard_Output_X7_7"}
	Module_4_Channel_3_Standard_Output_X7_7 AT %Q* : BOOL;
	{attribute addProperty Name "Module_4_Channel_4_Standard_Output_X7_8"}
	Module_4_Channel_4_Standard_Output_X7_8 AT %Q* : BOOL;
	{attribute addProperty Name "Module_5_Channel_1_Standard_Output_X9_1"}
	Module_5_Channel_1_Standard_Output_X9_1 AT %Q* : BOOL;
	{attribute addProperty Name "Module_5_Channel_2_Standard_Output_X9_2"}
	Module_5_Channel_2_Standard_Output_X9_2 AT %Q* : BOOL;
	{attribute addProperty Name "Module_5_Channel_3_Standard_Output_X9_3"}
	Module_5_Channel_3_Standard_Output_X9_3 AT %Q* : BOOL;
	{attribute addProperty Name "Module_5_Channel_4_Standard_Output_X9_4"}
	Module_5_Channel_4_Standard_Output_X9_4 AT %Q* : BOOL;
	{attribute addProperty Name "Module_6_Channel_1_Standard_Output_X9_5"}
	Module_6_Channel_1_Standard_Output_X9_5 AT %Q* : BOOL;
	{attribute addProperty Name "Module_6_Channel_2_Standard_Output_X9_6"}
	Module_6_Channel_2_Standard_Output_X9_6 AT %Q* : BOOL;
	{attribute addProperty Name "Module_6_Channel_3_Standard_Output_X9_7"}
	Module_6_Channel_3_Standard_Output_X9_7 AT %Q* : BOOL;
	{attribute addProperty Name "Module_6_Channel_4_Standard_Output_X9_8"}
	Module_6_Channel_4_Standard_Output_X9_8 AT %Q* : BOOL;
	{attribute addProperty Name "Relais_Module_Channel_1_Standard_Output_X4_1_X4_5"}
	Relais_Module_Channel_1_Standard_Output_X4_1_X4_5 AT %Q* : BOOL;
	{attribute addProperty Name "Relais_Module_Channel_2_Standard_Output_X4_2_X4_6"}
	Relais_Module_Channel_2_Standard_Output_X4_2_X4_6 AT %Q* : BOOL;
	{attribute addProperty Name "Relais_Module_Channel_3_Standard_Output_X4_3_X4_7"}
	Relais_Module_Channel_3_Standard_Output_X4_3_X4_7 AT %Q* : BOOL;
	{attribute addProperty Name "Relais_Module_Channel_4_Standard_Output_X4_4_X4_8"}
	Relais_Module_Channel_4_Standard_Output_X4_4_X4_8 AT %Q* : BOOL;
END_STRUCT
END_TYPE

// ---- DUTs/IO/PDOs/FSLOGIC_Inputs_EEE9388E.TcDUT
{attribute 'GeneratedUsingTerminal: EK1960-0000-0019'}
{attribute addProperty BoxType "EK1960-0000-0019"}
{attribute addProperty Id "Safe_Logic_StateAT %I*USINT1Cycle_CounterAT %I*USINT1"}
{attribute addProperty CRC "4008261774"}
{attribute addProperty Size "2"}
TYPE FSLOGIC_Inputs_EEE9388E EXTENDS InputBase_8311D824 :
STRUCT
	{attribute addProperty Name "Safe_Logic_State"}
	Safe_Logic_State AT %I* : USINT;
	{attribute addProperty Name "Cycle_Counter"}
	Cycle_Counter AT %I* : USINT;
END_STRUCT
END_TYPE

// ---- DUTs/IO/PDOs/EMPTY_STRUCTURE.TcDUT
{attribute 'GeneratedUsingTerminal: EK1960-0000-0019'}
{attribute addProperty BoxType "EK1960-0000-0019"}
{attribute addProperty Id "EMPTY_STRUCTURE"}
{attribute addProperty CRC "0"}
{attribute addProperty Size "0"}
TYPE EMPTY_STRUCTURE :
STRUCT
END_STRUCT
END_TYPE

// ---- DUTs/IO/PDOs/WcState_B516A264.TcDUT
{attribute 'GeneratedUsingTerminal: EK1960-0000-0019'}
{attribute addProperty BoxType "EK1960-0000-0019"}
{attribute addProperty Id "WcState0AT %I*BOOL1WcState1AT %I*BOOL1InputToggle0AT %I*BOOL1InputToggle1AT %I*BOOL1"}
{attribute addProperty CRC "3038159460"}
{attribute addProperty Size "4"}
TYPE WcState_B516A264 EXTENDS InputBase_8311D824 :
STRUCT
	{attribute addProperty Name "WcState0"}
	WcState0 AT %I* : BOOL;
	{attribute addProperty Name "WcState1"}
	WcState1 AT %I* : BOOL;
	{attribute addProperty Name "InputToggle0"}
	InputToggle0 AT %I* : BOOL;
	{attribute addProperty Name "InputToggle1"}
	InputToggle1 AT %I* : BOOL;
END_STRUCT
END_TYPE

// ---- DUTs/IO/PDOs/InfoData_32EB74EA.TcDUT
{attribute 'GeneratedUsingTerminal: EK1960-0000-0019'}
{attribute addProperty BoxType "EK1960-0000-0019"}
{attribute addProperty Id "AdsAddrAT %I*AMSADDR8StateAT %I*UINT2"}
{attribute addProperty CRC "854291690"}
{attribute addProperty Size "10"}
TYPE InfoData_32EB74EA EXTENDS InputBase_8311D824 :
STRUCT
	{attribute addProperty Name "AdsAddr"}
	AdsAddr AT %I* : AMSADDR;
	{attribute addProperty Name "State"}
	State AT %I* : UINT;
END_STRUCT
END_TYPE

// ---- DUTs/IO/PDOs/Module_1_FSoE_BE928FF7.TcDUT
{attribute 'GeneratedUsingTerminal: EK1960-0000-0019'}
{attribute addProperty BoxType "EK1960-0000-0019"}
{attribute addProperty Id "FSoE_InputsFSoE_Inputs_9283FC6947FSoE_OutputsFSoE_Outputs_79E75DAB51"}
{attribute addProperty CRC "3197276151"}
{attribute addProperty Size "98"}
TYPE Module_1_FSoE_BE928FF7 :
STRUCT
	{attribute addProperty Name "FSoE_Inputs"}
	FSoE_Inputs  : FSoE_Inputs_9283FC69;
	{attribute addProperty Name "FSoE_Outputs"}
	FSoE_Outputs  : FSoE_Outputs_79E75DAB;
END_STRUCT
END_TYPE

// ---- DUTs/IO/PDOs/Module_2_FSOUT_E84B1B00.TcDUT
{attribute 'GeneratedUsingTerminal: EK1960-0000-0019'}
{attribute addProperty BoxType "EK1960-0000-0019"}
{attribute addProperty Id "OutputsOutputs_63C46CC828"}
{attribute addProperty CRC "3897236224"}
{attribute addProperty Size "28"}
TYPE Module_2_FSOUT_E84B1B00 :
STRUCT
	{attribute addProperty Name "Outputs"}
	Outputs  : Outputs_63C46CC8;
END_STRUCT
END_TYPE

// ---- DUTs/IO/PDOs/Module_3_FSLOGIC_DEAB4522.TcDUT
{attribute 'GeneratedUsingTerminal: EK1960-0000-0019'}
{attribute addProperty BoxType "EK1960-0000-0019"}
{attribute addProperty Id "FSLOGIC_InputsFSLOGIC_Inputs_EEE9388E2FSLOGIC_OutputsEMPTY_STRUCTURE0"}
{attribute addProperty CRC "3735766306"}
{attribute addProperty Size "2"}
TYPE Module_3_FSLOGIC_DEAB4522 :
STRUCT
	{attribute addProperty Name "FSLOGIC_Inputs"}
	FSLOGIC_Inputs  : FSLOGIC_Inputs_EEE9388E;
	{attribute addProperty Name "FSLOGIC_Outputs"}
	FSLOGIC_Outputs  : EMPTY_STRUCTURE;
END_STRUCT
END_TYPE

// ---- DUTs/IO/PDOs/FSoE_Inputs_6CB74C4A.TcDUT
{attribute 'GeneratedUsingTerminal: EK1960-0000-0021'}
{attribute addProperty BoxType "EK1960-0000-0021"}
{attribute addProperty Id "FSOEAT %I*FSOE_39DE0EE047"}
{attribute addProperty CRC "1823951946"}
{attribute addProperty Size "47"}
TYPE FSoE_Inputs_6CB74C4A EXTENDS InputBase_8311D824 :
STRUCT
	{attribute addProperty Name "FSOE"}
	FSOE AT %I* : FSOE_39DE0EE0;
END_STRUCT
END_TYPE

// ---- DUTs/IO/PDOs/FSoE_Outputs_D8082339.TcDUT
{attribute 'GeneratedUsingTerminal: EK1960-0000-0021'}
{attribute addProperty BoxType "EK1960-0000-0021"}
{attribute addProperty Id "FSOEAT %Q*FSOE_3E4279E151"}
{attribute addProperty CRC "3624411961"}
{attribute addProperty Size "51"}
TYPE FSoE_Outputs_D8082339 EXTENDS OutputBase_10CEE7DE :
STRUCT
	{attribute addProperty Name "FSOE"}
	FSOE AT %Q* : FSOE_3E4279E1;
END_STRUCT
END_TYPE

// ---- DUTs/IO/PDOs/Outputs_D994E0F9.TcDUT
{attribute 'GeneratedUsingTerminal: EK1960-0000-0021'}
{attribute addProperty BoxType "EK1960-0000-0021"}
{attribute addProperty Id "Module_1_Channel_1_Standard_Output_X5_1AT %Q*BOOL1Module_1_Channel_2_Standard_Output_X5_2AT %Q*BOOL1Module_1_Channel_3_Standard_Output_X5_3AT %Q*BOOL1Module_1_Channel_4_Standard_Output_X5_4AT %Q*BOOL1Module_2_Channel_1_Standard_Output_X5_5AT %Q*BOOL1Module_2_Channel_2_Standard_Output_X5_6AT %Q*BOOL1Module_2_Channel_3_Standard_Output_X5_7AT %Q*BOOL1Module_2_Channel_4_Standard_Output_X5_8AT %Q*BOOL1Module_3_Channel_1_Standard_Output_X7_1AT %Q*BOOL1Module_3_Channel_2_Standard_Output_X7_2AT %Q*BOOL1Module_3_Channel_3_Standard_Output_X7_3AT %Q*BOOL1Module_3_Channel_4_Standard_Output_X7_4AT %Q*BOOL1Module_4_Channel_1_Standard_Output_X7_5AT %Q*BOOL1Module_4_Channel_2_Standard_Output_X7_6AT %Q*BOOL1Module_4_Channel_3_Standard_Output_X7_7AT %Q*BOOL1Module_4_Channel_4_Standard_Output_X7_8AT %Q*BOOL1Module_5_Channel_1_Standard_Output_X9_1AT %Q*BOOL1Module_5_Channel_2_Standard_Output_X9_2AT %Q*BOOL1Module_5_Channel_3_Standard_Output_X9_3AT %Q*BOOL1Module_5_Channel_4_Standard_Output_X9_4AT %Q*BOOL1Module_6_Channel_1_Standard_Output_X9_5AT %Q*BOOL1Module_6_Channel_2_Standard_Output_X9_6AT %Q*BOOL1Module_6_Channel_3_Standard_Output_X9_7AT %Q*BOOL1Module_6_Channel_4_Standard_Output_X9_8AT %Q*BOOL1"}
{attribute addProperty CRC "3650412793"}
{attribute addProperty Size "24"}
TYPE Outputs_D994E0F9 EXTENDS OutputBase_10CEE7DE :
STRUCT
	{attribute addProperty Name "Module_1_Channel_1_Standard_Output_X5_1"}
	Module_1_Channel_1_Standard_Output_X5_1 AT %Q* : BOOL;
	{attribute addProperty Name "Module_1_Channel_2_Standard_Output_X5_2"}
	Module_1_Channel_2_Standard_Output_X5_2 AT %Q* : BOOL;
	{attribute addProperty Name "Module_1_Channel_3_Standard_Output_X5_3"}
	Module_1_Channel_3_Standard_Output_X5_3 AT %Q* : BOOL;
	{attribute addProperty Name "Module_1_Channel_4_Standard_Output_X5_4"}
	Module_1_Channel_4_Standard_Output_X5_4 AT %Q* : BOOL;
	{attribute addProperty Name "Module_2_Channel_1_Standard_Output_X5_5"}
	Module_2_Channel_1_Standard_Output_X5_5 AT %Q* : BOOL;
	{attribute addProperty Name "Module_2_Channel_2_Standard_Output_X5_6"}
	Module_2_Channel_2_Standard_Output_X5_6 AT %Q* : BOOL;
	{attribute addProperty Name "Module_2_Channel_3_Standard_Output_X5_7"}
	Module_2_Channel_3_Standard_Output_X5_7 AT %Q* : BOOL;
	{attribute addProperty Name "Module_2_Channel_4_Standard_Output_X5_8"}
	Module_2_Channel_4_Standard_Output_X5_8 AT %Q* : BOOL;
	{attribute addProperty Name "Module_3_Channel_1_Standard_Output_X7_1"}
	Module_3_Channel_1_Standard_Output_X7_1 AT %Q* : BOOL;
	{attribute addProperty Name "Module_3_Channel_2_Standard_Output_X7_2"}
	Module_3_Channel_2_Standard_Output_X7_2 AT %Q* : BOOL;
	{attribute addProperty Name "Module_3_Channel_3_Standard_Output_X7_3"}
	Module_3_Channel_3_Standard_Output_X7_3 AT %Q* : BOOL;
	{attribute addProperty Name "Module_3_Channel_4_Standard_Output_X7_4"}
	Module_3_Channel_4_Standard_Output_X7_4 AT %Q* : BOOL;
	{attribute addProperty Name "Module_4_Channel_1_Standard_Output_X7_5"}
	Module_4_Channel_1_Standard_Output_X7_5 AT %Q* : BOOL;
	{attribute addProperty Name "Module_4_Channel_2_Standard_Output_X7_6"}
	Module_4_Channel_2_Standard_Output_X7_6 AT %Q* : BOOL;
	{attribute addProperty Name "Module_4_Channel_3_Standard_Output_X7_7"}
	Module_4_Channel_3_Standard_Output_X7_7 AT %Q* : BOOL;
	{attribute addProperty Name "Module_4_Channel_4_Standard_Output_X7_8"}
	Module_4_Channel_4_Standard_Output_X7_8 AT %Q* : BOOL;
	{attribute addProperty Name "Module_5_Channel_1_Standard_Output_X9_1"}
	Module_5_Channel_1_Standard_Output_X9_1 AT %Q* : BOOL;
	{attribute addProperty Name "Module_5_Channel_2_Standard_Output_X9_2"}
	Module_5_Channel_2_Standard_Output_X9_2 AT %Q* : BOOL;
	{attribute addProperty Name "Module_5_Channel_3_Standard_Output_X9_3"}
	Module_5_Channel_3_Standard_Output_X9_3 AT %Q* : BOOL;
	{attribute addProperty Name "Module_5_Channel_4_Standard_Output_X9_4"}
	Module_5_Channel_4_Standard_Output_X9_4 AT %Q* : BOOL;
	{attribute addProperty Name "Module_6_Channel_1_Standard_Output_X9_5"}
	Module_6_Channel_1_Standard_Output_X9_5 AT %Q* : BOOL;
	{attribute addProperty Name "Module_6_Channel_2_Standard_Output_X9_6"}
	Module_6_Channel_2_Standard_Output_X9_6 AT %Q* : BOOL;
	{attribute addProperty Name "Module_6_Channel_3_Standard_Output_X9_7"}
	Module_6_Channel_3_Standard_Output_X9_7 AT %Q* : BOOL;
	{attribute addProperty Name "Module_6_Channel_4_Standard_Output_X9_8"}
	Module_6_Channel_4_Standard_Output_X9_8 AT %Q* : BOOL;
END_STRUCT
END_TYPE

// ---- DUTs/IO/PDOs/Module_1_FSoE_042BAFD3.TcDUT
{attribute 'GeneratedUsingTerminal: EK1960-0000-0021'}
{attribute addProperty BoxType "EK1960-0000-0021"}
{attribute addProperty Id "FSoE_InputsFSoE_Inputs_6CB74C4A47FSoE_OutputsFSoE_Outputs_D808233951"}
{attribute addProperty CRC "69971923"}
{attribute addProperty Size "98"}
TYPE Module_1_FSoE_042BAFD3 :
STRUCT
	{attribute addProperty Name "FSoE_Inputs"}
	FSoE_Inputs  : FSoE_Inputs_6CB74C4A;
	{attribute addProperty Name "FSoE_Outputs"}
	FSoE_Outputs  : FSoE_Outputs_D8082339;
END_STRUCT
END_TYPE

// ---- DUTs/IO/PDOs/Module_2_FSOUT_8B7AA8A2.TcDUT
{attribute 'GeneratedUsingTerminal: EK1960-0000-0021'}
{attribute addProperty BoxType "EK1960-0000-0021"}
{attribute addProperty Id "OutputsOutputs_D994E0F924"}
{attribute addProperty CRC "2340071586"}
{attribute addProperty Size "24"}
TYPE Module_2_FSOUT_8B7AA8A2 :
STRUCT
	{attribute addProperty Name "Outputs"}
	Outputs  : Outputs_D994E0F9;
END_STRUCT
END_TYPE

// ---- DUTs/IO/PDOs/FSoE_Inputs_905C1934.TcDUT
{attribute 'GeneratedUsingTerminal: EK1960-2600-0019'}
{attribute addProperty BoxType "EK1960-2600-0019"}
{attribute addProperty Id "FSOEAT %I*FSOE_BAA7477B48"}
{attribute addProperty CRC "2421954868"}
{attribute addProperty Size "48"}
TYPE FSoE_Inputs_905C1934 EXTENDS InputBase_8311D824 :
STRUCT
	{attribute addProperty Name "FSOE"}
	FSOE AT %I* : FSOE_BAA7477B;
END_STRUCT
END_TYPE

// ---- DUTs/IO/PDOs/FSoE_Outputs_77F9785A.TcDUT
{attribute 'GeneratedUsingTerminal: EK1960-2600-0019'}
{attribute addProperty BoxType "EK1960-2600-0019"}
{attribute addProperty Id "FSOEAT %Q*FSOE_CEFF8C5656"}
{attribute addProperty CRC "2012837978"}
{attribute addProperty Size "56"}
TYPE FSoE_Outputs_77F9785A EXTENDS OutputBase_10CEE7DE :
STRUCT
	{attribute addProperty Name "FSOE"}
	FSOE AT %Q* : FSOE_CEFF8C56;
END_STRUCT
END_TYPE

// ---- DUTs/IO/PDOs/Module_1_FSoE_7E6C60DE.TcDUT
{attribute 'GeneratedUsingTerminal: EK1960-2600-0019'}
{attribute addProperty BoxType "EK1960-2600-0019"}
{attribute addProperty Id "FSoE_InputsFSoE_Inputs_905C193448FSoE_OutputsFSoE_Outputs_77F9785A56"}
{attribute addProperty CRC "2121031902"}
{attribute addProperty Size "104"}
TYPE Module_1_FSoE_7E6C60DE :
STRUCT
	{attribute addProperty Name "FSoE_Inputs"}
	FSoE_Inputs  : FSoE_Inputs_905C1934;
	{attribute addProperty Name "FSoE_Outputs"}
	FSoE_Outputs  : FSoE_Outputs_77F9785A;
END_STRUCT
END_TYPE

// ---- DUTs/IO/PDOs/FSoE_Inputs_A1F422BE.TcDUT
{attribute 'GeneratedUsingTerminal: EK1960-2600-0021'}
{attribute addProperty BoxType "EK1960-2600-0021"}
{attribute addProperty Id "FSOEAT %I*FSOE_E251F24448"}
{attribute addProperty CRC "2717131454"}
{attribute addProperty Size "48"}
TYPE FSoE_Inputs_A1F422BE EXTENDS InputBase_8311D824 :
STRUCT
	{attribute addProperty Name "FSOE"}
	FSOE AT %I* : FSOE_E251F244;
END_STRUCT
END_TYPE

// ---- DUTs/IO/PDOs/FSoE_Outputs_37DEC564.TcDUT
{attribute 'GeneratedUsingTerminal: EK1960-2600-0021'}
{attribute addProperty BoxType "EK1960-2600-0021"}
{attribute addProperty Id "FSOEAT %Q*FSOE_CDFABDDF56"}
{attribute addProperty CRC "937346404"}
{attribute addProperty Size "56"}
TYPE FSoE_Outputs_37DEC564 EXTENDS OutputBase_10CEE7DE :
STRUCT
	{attribute addProperty Name "FSOE"}
	FSOE AT %Q* : FSOE_CDFABDDF;
END_STRUCT
END_TYPE

// ---- DUTs/IO/PDOs/Module_1_FSoE_B78AD590.TcDUT
{attribute 'GeneratedUsingTerminal: EK1960-2600-0021'}
{attribute addProperty BoxType "EK1960-2600-0021"}
{attribute addProperty Id "FSoE_InputsFSoE_Inputs_A1F422BE48FSoE_OutputsFSoE_Outputs_37DEC56456"}
{attribute addProperty CRC "3079329168"}
{attribute addProperty Size "104"}
TYPE Module_1_FSoE_B78AD590 :
STRUCT
	{attribute addProperty Name "FSoE_Inputs"}
	FSoE_Inputs  : FSoE_Inputs_A1F422BE;
	{attribute addProperty Name "FSoE_Outputs"}
	FSoE_Outputs  : FSoE_Outputs_37DEC564;
END_STRUCT
END_TYPE

// ---- DUTs/IO/PDOs/InfoData_E68C61CD.TcDUT
{attribute 'GeneratedUsingTerminal: IODEVICETYPE_ETHERCATPROT'}
{attribute addProperty BoxType "IODEVICETYPE_ETHERCATPROT"}
{attribute addProperty Id "ChangeCountAT %I*UINT2DevIdAT %I*UINT2AmsNetIdAT %I*AMSNETID6CfgSlaveCountAT %I*UINT2DcToTcTimeOffsetAT %I*LINT8DcToExtTimeOffsetAT %I*LINT8"}
{attribute addProperty CRC "3867959757"}
{attribute addProperty Size "28"}
TYPE InfoData_E68C61CD EXTENDS InputBase_8311D824 :
STRUCT
	{attribute addProperty Name "ChangeCount"}
	ChangeCount AT %I* : UINT;
	{attribute addProperty Name "DevId"}
	DevId AT %I* : UINT;
	{attribute addProperty Name "AmsNetId"}
	AmsNetId AT %I* : AMSNETID;
	{attribute addProperty Name "CfgSlaveCount"}
	CfgSlaveCount AT %I* : UINT;
	{attribute addProperty Name "DcToTcTimeOffset"}
	DcToTcTimeOffset AT %I* : LINT;
	{attribute addProperty Name "DcToExtTimeOffset"}
	DcToExtTimeOffset AT %I* : LINT;
END_STRUCT
END_TYPE

// ---- DUTs/IO/PDOs/InfoData_2A97D6CF.TcDUT
{attribute 'GeneratedUsingTerminal: IODEVICETYPE_ETHERCATPROT'}
{attribute addProperty BoxType "IODEVICETYPE_ETHERCATPROT"}
{attribute addProperty Id "ObjectIdAT %I*OTCID4StateAT %I*UINT2SlaveCountAT %I*UINT2"}
{attribute addProperty CRC "714593999"}
{attribute addProperty Size "8"}
TYPE InfoData_2A97D6CF EXTENDS InputBase_8311D824 :
STRUCT
	{attribute addProperty Name "ObjectId"}
	ObjectId AT %I* : OTCID;
	{attribute addProperty Name "State"}
	State AT %I* : UINT;
	{attribute addProperty Name "SlaveCount"}
	SlaveCount AT %I* : UINT;
END_STRUCT
END_TYPE

// ---- DUTs/IO/PDOs/Inputs_25A0042B.TcDUT
{attribute 'GeneratedUsingTerminal: IODEVICETYPE_ETHERCATPROT'}
{attribute addProperty BoxType "IODEVICETYPE_ETHERCATPROT"}
{attribute addProperty Id "SlaveCountAT %I*UINT2DevStateAT %I*UINT2Frm0StateAT %I*UINT2Frm0WcStateAT %I*UINT2Frm0InputToggleAT %I*UINT2Frm1StateAT %I*UINT2Frm1WcStateAT %I*UINT2Frm1InputToggleAT %I*UINT2Frm2StateAT %I*UINT2Frm2WcStateAT %I*UINT2Frm2InputToggleAT %I*UINT2Frm3StateAT %I*UINT2Frm3WcStateAT %I*UINT2Frm3InputToggleAT %I*UINT2Frm4StateAT %I*UINT2Frm4WcStateAT %I*UINT2Frm4InputToggleAT %I*UINT2Frm5StateAT %I*UINT2Frm5WcStateAT %I*UINT2Frm5InputToggleAT %I*UINT2Frm6StateAT %I*UINT2Frm6WcStateAT %I*UINT2Frm6InputToggleAT %I*UINT2Frm7StateAT %I*UINT2Frm7WcStateAT %I*UINT2Frm7InputToggleAT %I*UINT2Frm8StateAT %I*UINT2Frm8WcStateAT %I*UINT2Frm8InputToggleAT %I*UINT2Frm9StateAT %I*UINT2Frm9WcStateAT %I*UINT2Frm9InputToggleAT %I*UINT2Frm10StateAT %I*UINT2Frm10WcStateAT %I*UINT2Frm10InputToggleAT %I*UINT2Frm11StateAT %I*UINT2Frm11WcStateAT %I*UINT2Frm11InputToggleAT %I*UINT2Frm12StateAT %I*UINT2Frm12WcStateAT %I*UINT2Frm12InputToggleAT %I*UINT2Frm13StateAT %I*UINT2Frm13WcStateAT %I*UINT2Frm13InputToggleAT %I*UINT2Frm14StateAT %I*UINT2Frm14WcStateAT %I*UINT2Frm14InputToggleAT %I*UINT2Frm15StateAT %I*UINT2Frm15WcStateAT %I*UINT2Frm15InputToggleAT %I*UINT2Frm16StateAT %I*UINT2Frm16WcStateAT %I*UINT2Frm16InputToggleAT %I*UINT2Frm17StateAT %I*UINT2Frm17WcStateAT %I*UINT2Frm17InputToggleAT %I*UINT2Frm18StateAT %I*UINT2Frm18WcStateAT %I*UINT2Frm18InputToggleAT %I*UINT2Frm19StateAT %I*UINT2Frm19WcStateAT %I*UINT2Frm19InputToggleAT %I*UINT2Frm20StateAT %I*UINT2Frm20WcStateAT %I*UINT2Frm20InputToggleAT %I*UINT2Frm21StateAT %I*UINT2Frm21WcStateAT %I*UINT2Frm21InputToggleAT %I*UINT2Frm22StateAT %I*UINT2Frm22WcStateAT %I*UINT2Frm22InputToggleAT %I*UINT2Frm23StateAT %I*UINT2Frm23WcStateAT %I*UINT2Frm23InputToggleAT %I*UINT2Frm24StateAT %I*UINT2Frm24WcStateAT %I*UINT2Frm24InputToggleAT %I*UINT2Frm25StateAT %I*UINT2Frm25WcStateAT %I*UINT2Frm25InputToggleAT %I*UINT2"}
{attribute addProperty CRC "631243819"}
{attribute addProperty Size "160"}
TYPE Inputs_25A0042B EXTENDS InputBase_8311D824 :
STRUCT
	{attribute addProperty Name "SlaveCount"}
	SlaveCount AT %I* : UINT;
	{attribute addProperty Name "DevState"}
	DevState AT %I* : UINT;
	{attribute addProperty Name "Frm0State"}
	Frm0State AT %I* : UINT;
	{attribute addProperty Name "Frm0WcState"}
	Frm0WcState AT %I* : UINT;
	{attribute addProperty Name "Frm0InputToggle"}
	Frm0InputToggle AT %I* : UINT;
	{attribute addProperty Name "Frm1State"}
	Frm1State AT %I* : UINT;
	{attribute addProperty Name "Frm1WcState"}
	Frm1WcState AT %I* : UINT;
	{attribute addProperty Name "Frm1InputToggle"}
	Frm1InputToggle AT %I* : UINT;
	{attribute addProperty Name "Frm2State"}
	Frm2State AT %I* : UINT;
	{attribute addProperty Name "Frm2WcState"}
	Frm2WcState AT %I* : UINT;
	{attribute addProperty Name "Frm2InputToggle"}
	Frm2InputToggle AT %I* : UINT;
	{attribute addProperty Name "Frm3State"}
	Frm3State AT %I* : UINT;
	{attribute addProperty Name "Frm3WcState"}
	Frm3WcState AT %I* : UINT;
	{attribute addProperty Name "Frm3InputToggle"}
	Frm3InputToggle AT %I* : UINT;
	{attribute addProperty Name "Frm4State"}
	Frm4State AT %I* : UINT;
	{attribute addProperty Name "Frm4WcState"}
	Frm4WcState AT %I* : UINT;
	{attribute addProperty Name "Frm4InputToggle"}
	Frm4InputToggle AT %I* : UINT;
	{attribute addProperty Name "Frm5State"}
	Frm5State AT %I* : UINT;
	{attribute addProperty Name "Frm5WcState"}
	Frm5WcState AT %I* : UINT;
	{attribute addProperty Name "Frm5InputToggle"}
	Frm5InputToggle AT %I* : UINT;
	{attribute addProperty Name "Frm6State"}
	Frm6State AT %I* : UINT;
	{attribute addProperty Name "Frm6WcState"}
	Frm6WcState AT %I* : UINT;
	{attribute addProperty Name "Frm6InputToggle"}
	Frm6InputToggle AT %I* : UINT;
	{attribute addProperty Name "Frm7State"}
	Frm7State AT %I* : UINT;
	{attribute addProperty Name "Frm7WcState"}
	Frm7WcState AT %I* : UINT;
	{attribute addProperty Name "Frm7InputToggle"}
	Frm7InputToggle AT %I* : UINT;
	{attribute addProperty Name "Frm8State"}
	Frm8State AT %I* : UINT;
	{attribute addProperty Name "Frm8WcState"}
	Frm8WcState AT %I* : UINT;
	{attribute addProperty Name "Frm8InputToggle"}
	Frm8InputToggle AT %I* : UINT;
	{attribute addProperty Name "Frm9State"}
	Frm9State AT %I* : UINT;
	{attribute addProperty Name "Frm9WcState"}
	Frm9WcState AT %I* : UINT;
	{attribute addProperty Name "Frm9InputToggle"}
	Frm9InputToggle AT %I* : UINT;
	{attribute addProperty Name "Frm10State"}
	Frm10State AT %I* : UINT;
	{attribute addProperty Name "Frm10WcState"}
	Frm10WcState AT %I* : UINT;
	{attribute addProperty Name "Frm10InputToggle"}
	Frm10InputToggle AT %I* : UINT;
	{attribute addProperty Name "Frm11State"}
	Frm11State AT %I* : UINT;
	{attribute addProperty Name "Frm11WcState"}
	Frm11WcState AT %I* : UINT;
	{attribute addProperty Name "Frm11InputToggle"}
	Frm11InputToggle AT %I* : UINT;
	{attribute addProperty Name "Frm12State"}
	Frm12State AT %I* : UINT;
	{attribute addProperty Name "Frm12WcState"}
	Frm12WcState AT %I* : UINT;
	{attribute addProperty Name "Frm12InputToggle"}
	Frm12InputToggle AT %I* : UINT;
	{attribute addProperty Name "Frm13State"}
	Frm13State AT %I* : UINT;
	{attribute addProperty Name "Frm13WcState"}
	Frm13WcState AT %I* : UINT;
	{attribute addProperty Name "Frm13InputToggle"}
	Frm13InputToggle AT %I* : UINT;
	{attribute addProperty Name "Frm14State"}
	Frm14State AT %I* : UINT;
	{attribute addProperty Name "Frm14WcState"}
	Frm14WcState AT %I* : UINT;
	{attribute addProperty Name "Frm14InputToggle"}
	Frm14InputToggle AT %I* : UINT;
	{attribute addProperty Name "Frm15State"}
	Frm15State AT %I* : UINT;
	{attribute addProperty Name "Frm15WcState"}
	Frm15WcState AT %I* : UINT;
	{attribute addProperty Name "Frm15InputToggle"}
	Frm15InputToggle AT %I* : UINT;
	{attribute addProperty Name "Frm16State"}
	Frm16State AT %I* : UINT;
	{attribute addProperty Name "Frm16WcState"}
	Frm16WcState AT %I* : UINT;
	{attribute addProperty Name "Frm16InputToggle"}
	Frm16InputToggle AT %I* : UINT;
	{attribute addProperty Name "Frm17State"}
	Frm17State AT %I* : UINT;
	{attribute addProperty Name "Frm17WcState"}
	Frm17WcState AT %I* : UINT;
	{attribute addProperty Name "Frm17InputToggle"}
	Frm17InputToggle AT %I* : UINT;
	{attribute addProperty Name "Frm18State"}
	Frm18State AT %I* : UINT;
	{attribute addProperty Name "Frm18WcState"}
	Frm18WcState AT %I* : UINT;
	{attribute addProperty Name "Frm18InputToggle"}
	Frm18InputToggle AT %I* : UINT;
	{attribute addProperty Name "Frm19State"}
	Frm19State AT %I* : UINT;
	{attribute addProperty Name "Frm19WcState"}
	Frm19WcState AT %I* : UINT;
	{attribute addProperty Name "Frm19InputToggle"}
	Frm19InputToggle AT %I* : UINT;
	{attribute addProperty Name "Frm20State"}
	Frm20State AT %I* : UINT;
	{attribute addProperty Name "Frm20WcState"}
	Frm20WcState AT %I* : UINT;
	{attribute addProperty Name "Frm20InputToggle"}
	Frm20InputToggle AT %I* : UINT;
	{attribute addProperty Name "Frm21State"}
	Frm21State AT %I* : UINT;
	{attribute addProperty Name "Frm21WcState"}
	Frm21WcState AT %I* : UINT;
	{attribute addProperty Name "Frm21InputToggle"}
	Frm21InputToggle AT %I* : UINT;
	{attribute addProperty Name "Frm22State"}
	Frm22State AT %I* : UINT;
	{attribute addProperty Name "Frm22WcState"}
	Frm22WcState AT %I* : UINT;
	{attribute addProperty Name "Frm22InputToggle"}
	Frm22InputToggle AT %I* : UINT;
	{attribute addProperty Name "Frm23State"}
	Frm23State AT %I* : UINT;
	{attribute addProperty Name "Frm23WcState"}
	Frm23WcState AT %I* : UINT;
	{attribute addProperty Name "Frm23InputToggle"}
	Frm23InputToggle AT %I* : UINT;
	{attribute addProperty Name "Frm24State"}
	Frm24State AT %I* : UINT;
	{attribute addProperty Name "Frm24WcState"}
	Frm24WcState AT %I* : UINT;
	{attribute addProperty Name "Frm24InputToggle"}
	Frm24InputToggle AT %I* : UINT;
	{attribute addProperty Name "Frm25State"}
	Frm25State AT %I* : UINT;
	{attribute addProperty Name "Frm25WcState"}
	Frm25WcState AT %I* : UINT;
	{attribute addProperty Name "Frm25InputToggle"}
	Frm25InputToggle AT %I* : UINT;
END_STRUCT
END_TYPE

// ---- DUTs/IO/PDOs/Outputs_2397A10E.TcDUT
{attribute 'GeneratedUsingTerminal: IODEVICETYPE_ETHERCATPROT'}
{attribute addProperty BoxType "IODEVICETYPE_ETHERCATPROT"}
{attribute addProperty Id "DevCtrlAT %Q*UINT2Frm0CtrlAT %Q*UINT2Frm0WcCtrlAT %Q*UINT2Frm1CtrlAT %Q*UINT2Frm1WcCtrlAT %Q*UINT2Frm2CtrlAT %Q*UINT2Frm2WcCtrlAT %Q*UINT2Frm3CtrlAT %Q*UINT2Frm3WcCtrlAT %Q*UINT2Frm4CtrlAT %Q*UINT2Frm4WcCtrlAT %Q*UINT2Frm5CtrlAT %Q*UINT2Frm5WcCtrlAT %Q*UINT2Frm6CtrlAT %Q*UINT2Frm6WcCtrlAT %Q*UINT2Frm7CtrlAT %Q*UINT2Frm7WcCtrlAT %Q*UINT2Frm8CtrlAT %Q*UINT2Frm8WcCtrlAT %Q*UINT2Frm9CtrlAT %Q*UINT2Frm9WcCtrlAT %Q*UINT2Frm10CtrlAT %Q*UINT2Frm10WcCtrlAT %Q*UINT2Frm11CtrlAT %Q*UINT2Frm11WcCtrlAT %Q*UINT2Frm12CtrlAT %Q*UINT2Frm12WcCtrlAT %Q*UINT2Frm13CtrlAT %Q*UINT2Frm13WcCtrlAT %Q*UINT2Frm14CtrlAT %Q*UINT2Frm14WcCtrlAT %Q*UINT2Frm15CtrlAT %Q*UINT2Frm15WcCtrlAT %Q*UINT2Frm16CtrlAT %Q*UINT2Frm16WcCtrlAT %Q*UINT2Frm17CtrlAT %Q*UINT2Frm17WcCtrlAT %Q*UINT2Frm18CtrlAT %Q*UINT2Frm18WcCtrlAT %Q*UINT2Frm19CtrlAT %Q*UINT2Frm19WcCtrlAT %Q*UINT2Frm20CtrlAT %Q*UINT2Frm20WcCtrlAT %Q*UINT2Frm21CtrlAT %Q*UINT2Frm21WcCtrlAT %Q*UINT2Frm22CtrlAT %Q*UINT2Frm22WcCtrlAT %Q*UINT2Frm23CtrlAT %Q*UINT2Frm23WcCtrlAT %Q*UINT2Frm24CtrlAT %Q*UINT2Frm24WcCtrlAT %Q*UINT2Frm25CtrlAT %Q*UINT2Frm25WcCtrlAT %Q*UINT2"}
{attribute addProperty CRC "597139726"}
{attribute addProperty Size "106"}
TYPE Outputs_2397A10E EXTENDS OutputBase_10CEE7DE :
STRUCT
	{attribute addProperty Name "DevCtrl"}
	DevCtrl AT %Q* : UINT;
	{attribute addProperty Name "Frm0Ctrl"}
	Frm0Ctrl AT %Q* : UINT;
	{attribute addProperty Name "Frm0WcCtrl"}
	Frm0WcCtrl AT %Q* : UINT;
	{attribute addProperty Name "Frm1Ctrl"}
	Frm1Ctrl AT %Q* : UINT;
	{attribute addProperty Name "Frm1WcCtrl"}
	Frm1WcCtrl AT %Q* : UINT;
	{attribute addProperty Name "Frm2Ctrl"}
	Frm2Ctrl AT %Q* : UINT;
	{attribute addProperty Name "Frm2WcCtrl"}
	Frm2WcCtrl AT %Q* : UINT;
	{attribute addProperty Name "Frm3Ctrl"}
	Frm3Ctrl AT %Q* : UINT;
	{attribute addProperty Name "Frm3WcCtrl"}
	Frm3WcCtrl AT %Q* : UINT;
	{attribute addProperty Name "Frm4Ctrl"}
	Frm4Ctrl AT %Q* : UINT;
	{attribute addProperty Name "Frm4WcCtrl"}
	Frm4WcCtrl AT %Q* : UINT;
	{attribute addProperty Name "Frm5Ctrl"}
	Frm5Ctrl AT %Q* : UINT;
	{attribute addProperty Name "Frm5WcCtrl"}
	Frm5WcCtrl AT %Q* : UINT;
	{attribute addProperty Name "Frm6Ctrl"}
	Frm6Ctrl AT %Q* : UINT;
	{attribute addProperty Name "Frm6WcCtrl"}
	Frm6WcCtrl AT %Q* : UINT;
	{attribute addProperty Name "Frm7Ctrl"}
	Frm7Ctrl AT %Q* : UINT;
	{attribute addProperty Name "Frm7WcCtrl"}
	Frm7WcCtrl AT %Q* : UINT;
	{attribute addProperty Name "Frm8Ctrl"}
	Frm8Ctrl AT %Q* : UINT;
	{attribute addProperty Name "Frm8WcCtrl"}
	Frm8WcCtrl AT %Q* : UINT;
	{attribute addProperty Name "Frm9Ctrl"}
	Frm9Ctrl AT %Q* : UINT;
	{attribute addProperty Name "Frm9WcCtrl"}
	Frm9WcCtrl AT %Q* : UINT;
	{attribute addProperty Name "Frm10Ctrl"}
	Frm10Ctrl AT %Q* : UINT;
	{attribute addProperty Name "Frm10WcCtrl"}
	Frm10WcCtrl AT %Q* : UINT;
	{attribute addProperty Name "Frm11Ctrl"}
	Frm11Ctrl AT %Q* : UINT;
	{attribute addProperty Name "Frm11WcCtrl"}
	Frm11WcCtrl AT %Q* : UINT;
	{attribute addProperty Name "Frm12Ctrl"}
	Frm12Ctrl AT %Q* : UINT;
	{attribute addProperty Name "Frm12WcCtrl"}
	Frm12WcCtrl AT %Q* : UINT;
	{attribute addProperty Name "Frm13Ctrl"}
	Frm13Ctrl AT %Q* : UINT;
	{attribute addProperty Name "Frm13WcCtrl"}
	Frm13WcCtrl AT %Q* : UINT;
	{attribute addProperty Name "Frm14Ctrl"}
	Frm14Ctrl AT %Q* : UINT;
	{attribute addProperty Name "Frm14WcCtrl"}
	Frm14WcCtrl AT %Q* : UINT;
	{attribute addProperty Name "Frm15Ctrl"}
	Frm15Ctrl AT %Q* : UINT;
	{attribute addProperty Name "Frm15WcCtrl"}
	Frm15WcCtrl AT %Q* : UINT;
	{attribute addProperty Name "Frm16Ctrl"}
	Frm16Ctrl AT %Q* : UINT;
	{attribute addProperty Name "Frm16WcCtrl"}
	Frm16WcCtrl AT %Q* : UINT;
	{attribute addProperty Name "Frm17Ctrl"}
	Frm17Ctrl AT %Q* : UINT;
	{attribute addProperty Name "Frm17WcCtrl"}
	Frm17WcCtrl AT %Q* : UINT;
	{attribute addProperty Name "Frm18Ctrl"}
	Frm18Ctrl AT %Q* : UINT;
	{attribute addProperty Name "Frm18WcCtrl"}
	Frm18WcCtrl AT %Q* : UINT;
	{attribute addProperty Name "Frm19Ctrl"}
	Frm19Ctrl AT %Q* : UINT;
	{attribute addProperty Name "Frm19WcCtrl"}
	Frm19WcCtrl AT %Q* : UINT;
	{attribute addProperty Name "Frm20Ctrl"}
	Frm20Ctrl AT %Q* : UINT;
	{attribute addProperty Name "Frm20WcCtrl"}
	Frm20WcCtrl AT %Q* : UINT;
	{attribute addProperty Name "Frm21Ctrl"}
	Frm21Ctrl AT %Q* : UINT;
	{attribute addProperty Name "Frm21WcCtrl"}
	Frm21WcCtrl AT %Q* : UINT;
	{attribute addProperty Name "Frm22Ctrl"}
	Frm22Ctrl AT %Q* : UINT;
	{attribute addProperty Name "Frm22WcCtrl"}
	Frm22WcCtrl AT %Q* : UINT;
	{attribute addProperty Name "Frm23Ctrl"}
	Frm23Ctrl AT %Q* : UINT;
	{attribute addProperty Name "Frm23WcCtrl"}
	Frm23WcCtrl AT %Q* : UINT;
	{attribute addProperty Name "Frm24Ctrl"}
	Frm24Ctrl AT %Q* : UINT;
	{attribute addProperty Name "Frm24WcCtrl"}
	Frm24WcCtrl AT %Q* : UINT;
	{attribute addProperty Name "Frm25Ctrl"}
	Frm25Ctrl AT %Q* : UINT;
	{attribute addProperty Name "Frm25WcCtrl"}
	Frm25WcCtrl AT %Q* : UINT;
END_STRUCT
END_TYPE

// ---- DUTs/IO/Boxes/EK1100_1FC0878B.TcDUT
{attribute 'GeneratedUsingTerminal: EK1100-0000-0018'}
{attribute addProperty BoxType "EK1100-0000-0018"}
{attribute addProperty Description "EK1100 EtherCAT Coupler (2A E-Bus)"}
{attribute addProperty Physics "YKY"}
{attribute addProperty Id "InfoDataAT %I*InfoData_6F19DB2B2"}
{attribute addProperty CRC "532711307"}
{attribute addProperty Size "2"}
TYPE EK1100_1FC0878B EXTENDS EtcSlaveBoxBase_77A0E4A7 :
STRUCT
	{attribute addProperty Name "InfoData"}
	InfoData : InfoData_6F19DB2B;
END_STRUCT
END_TYPE

// ---- DUTs/IO/Boxes/EK1122_1FC0878B.TcDUT
{attribute 'GeneratedUsingTerminal: EK1122-0000-0018'}
{attribute addProperty BoxType "EK1122-0000-0018"}
{attribute addProperty Description "EK1122 2 port EtherCAT junction"}
{attribute addProperty Physics "KYKY"}
{attribute addProperty Id "InfoDataAT %I*InfoData_6F19DB2B2"}
{attribute addProperty CRC "532711307"}
{attribute addProperty Size "2"}
TYPE EK1122_1FC0878B EXTENDS EtcSlaveTerminalBase_947E5A46 :
STRUCT
	{attribute addProperty Name "InfoData"}
	InfoData : InfoData_6F19DB2B;
END_STRUCT
END_TYPE

// ---- DUTs/IO/Boxes/EK1101_957D888F.TcDUT
{attribute 'GeneratedUsingTerminal: EK1101-0000-0016'}
{attribute addProperty BoxType "EK1101-0000-0016"}
{attribute addProperty Description "EK1101 EtherCAT Coupler (2A E-Bus, ID switch)"}
{attribute addProperty Physics "YKY"}
{attribute addProperty Id "IDAT %I*ID_07C9D28F2WcStateAT %I*WcState_9091E0EB2InfoDataAT %I*InfoData_6F19DB2B2"}
{attribute addProperty CRC "2508032143"}
{attribute addProperty Size "6"}
TYPE EK1101_957D888F EXTENDS EtcSlaveBoxBase_77A0E4A7 :
STRUCT
	{attribute addProperty Name "ID"}
	ID : ID_07C9D28F;
	{attribute addProperty Name "WcState"}
	WcState : WcState_9091E0EB;
	{attribute addProperty Name "InfoData"}
	InfoData : InfoData_6F19DB2B;
END_STRUCT
END_TYPE

// ---- DUTs/IO/Boxes/EK1110_1FC0878B.TcDUT
{attribute 'GeneratedUsingTerminal: EK1110-0043-0016'}
{attribute addProperty BoxType "EK1110-0043-0016"}
{attribute addProperty Description "EK1110-0043 EtherCAT EJ coupler"}
{attribute addProperty Physics "KK"}
{attribute addProperty Id "InfoDataAT %I*InfoData_6F19DB2B2"}
{attribute addProperty CRC "532711307"}
{attribute addProperty Size "2"}
TYPE EK1110_1FC0878B EXTENDS EtcSlaveTerminalBase_947E5A46 :
STRUCT
	{attribute addProperty Name "InfoData"}
	InfoData : InfoData_6F19DB2B;
END_STRUCT
END_TYPE

// ---- DUTs/IO/Boxes/EK1121_1FC0878B.TcDUT
{attribute 'GeneratedUsingTerminal: EK1121-0010-0016'}
{attribute addProperty BoxType "EK1121-0010-0016"}
{attribute addProperty Description "EK1121-0010 1 port EtherCAT junction (Extended Distance)"}
{attribute addProperty Physics "K_KY"}
{attribute addProperty Id "InfoDataAT %I*InfoData_6F19DB2B2"}
{attribute addProperty CRC "532711307"}
{attribute addProperty Size "2"}
TYPE EK1121_1FC0878B EXTENDS EtcSlaveTerminalBase_947E5A46 :
STRUCT
	{attribute addProperty Name "InfoData"}
	InfoData : InfoData_6F19DB2B;
END_STRUCT
END_TYPE

// ---- DUTs/IO/Boxes/EK1200_013D0B49.TcDUT
{attribute 'GeneratedUsingTerminal: EK1200-1b58-0000'}
{attribute addProperty BoxType "EK1200-1b58-0000"}
{attribute addProperty Description "EK1200-7000 EtherCAT Power supply (1,5A E-Bus)"}
{attribute addProperty Physics "YK"}
{attribute addProperty Id "EK1200"}
{attribute addProperty CRC "20777801"}
{attribute addProperty Size "0"}
TYPE EK1200_013D0B49 EXTENDS EtcSlaveBoxBase_77A0E4A7 :
STRUCT
END_STRUCT
END_TYPE

// ---- DUTs/IO/Boxes/EK1300_6BC01D14.TcDUT
{attribute 'GeneratedUsingTerminal: EK1300-0000-0017'}
{attribute addProperty BoxType "EK1300-0000-0017"}
{attribute addProperty Description "EK1300 EtherCAT P Coupler (2A E-Bus)"}
{attribute addProperty Physics "YKY"}
{attribute addProperty Id "Status_UsAT %I*Status_Us_B1E819A21Status_UpAT %I*Status_Up_B1E819A21WcStateAT %I*WcState_9091E0EB2InfoDataAT %I*InfoData_6F19DB2B2"}
{attribute addProperty CRC "1807752468"}
{attribute addProperty Size "6"}
TYPE EK1300_6BC01D14 EXTENDS EtcSlaveBoxBase_77A0E4A7 :
STRUCT
	{attribute addProperty Name "Status_Us"}
	Status_Us : Status_Us_B1E819A2;
	{attribute addProperty Name "Status_Up"}
	Status_Up : Status_Up_B1E819A2;
	{attribute addProperty Name "WcState"}
	WcState : WcState_9091E0EB;
	{attribute addProperty Name "InfoData"}
	InfoData : InfoData_6F19DB2B;
END_STRUCT
END_TYPE

// ---- DUTs/IO/Boxes/EK1322_6BC01D14.TcDUT
{attribute 'GeneratedUsingTerminal: EK1322-0000-0017'}
{attribute addProperty BoxType "EK1322-0000-0017"}
{attribute addProperty Description "EK1322 2-port EtherCAT P junction with feed-in"}
{attribute addProperty Physics "KYKY"}
{attribute addProperty Id "Status_UsAT %I*Status_Us_B1E819A21Status_UpAT %I*Status_Up_B1E819A21WcStateAT %I*WcState_9091E0EB2InfoDataAT %I*InfoData_6F19DB2B2"}
{attribute addProperty CRC "1807752468"}
{attribute addProperty Size "6"}
TYPE EK1322_6BC01D14 EXTENDS EtcSlaveTerminalBase_947E5A46 :
STRUCT
	{attribute addProperty Name "Status_Us"}
	Status_Us : Status_Us_B1E819A2;
	{attribute addProperty Name "Status_Up"}
	Status_Up : Status_Up_B1E819A2;
	{attribute addProperty Name "WcState"}
	WcState : WcState_9091E0EB;
	{attribute addProperty Name "InfoData"}
	InfoData : InfoData_6F19DB2B;
END_STRUCT
END_TYPE

// ---- DUTs/IO/Boxes/EK1310_6BC01D14.TcDUT
{attribute 'GeneratedUsingTerminal: EK1310-0000-0017'}
{attribute addProperty BoxType "EK1310-0000-0017"}
{attribute addProperty Description "EK1310 EtherCAT P extension with feed-in"}
{attribute addProperty Physics "KY"}
{attribute addProperty Id "Status_UsAT %I*Status_Us_B1E819A21Status_UpAT %I*Status_Up_B1E819A21WcStateAT %I*WcState_9091E0EB2InfoDataAT %I*InfoData_6F19DB2B2"}
{attribute addProperty CRC "1807752468"}
{attribute addProperty Size "6"}
TYPE EK1310_6BC01D14 EXTENDS EtcSlaveTerminalBase_947E5A46 :
STRUCT
	{attribute addProperty Name "Status_Us"}
	Status_Us : Status_Us_B1E819A2;
	{attribute addProperty Name "Status_Up"}
	Status_Up : Status_Up_B1E819A2;
	{attribute addProperty Name "WcState"}
	WcState : WcState_9091E0EB;
	{attribute addProperty Name "InfoData"}
	InfoData : InfoData_6F19DB2B;
END_STRUCT
END_TYPE

// ---- DUTs/IO/Boxes/EK1501_957D888F.TcDUT
{attribute 'GeneratedUsingTerminal: EK1501-0000-0016'}
{attribute addProperty BoxType "EK1501-0000-0016"}
{attribute addProperty Description "EK1501 EtherCAT Coupler (2A E-Bus, FX-MultiMode, ID switch)"}
{attribute addProperty Physics "YKY"}
{attribute addProperty Id "IDAT %I*ID_07C9D28F2WcStateAT %I*WcState_9091E0EB2InfoDataAT %I*InfoData_6F19DB2B2"}
{attribute addProperty CRC "2508032143"}
{attribute addProperty Size "6"}
TYPE EK1501_957D888F EXTENDS EtcSlaveBoxBase_77A0E4A7 :
STRUCT
	{attribute addProperty Name "ID"}
	ID : ID_07C9D28F;
	{attribute addProperty Name "WcState"}
	WcState : WcState_9091E0EB;
	{attribute addProperty Name "InfoData"}
	InfoData : InfoData_6F19DB2B;
END_STRUCT
END_TYPE

// ---- DUTs/IO/Boxes/EK1541_957D888F.TcDUT
{attribute 'GeneratedUsingTerminal: EK1541-0000-0016'}
{attribute addProperty BoxType "EK1541-0000-0016"}
{attribute addProperty Description "EK1541 EtherCAT Coupler (2A E-Bus, POF, ID switch)"}
{attribute addProperty Physics "YKY"}
{attribute addProperty Id "IDAT %I*ID_07C9D28F2WcStateAT %I*WcState_9091E0EB2InfoDataAT %I*InfoData_6F19DB2B2"}
{attribute addProperty CRC "2508032143"}
{attribute addProperty Size "6"}
TYPE EK1541_957D888F EXTENDS EtcSlaveBoxBase_77A0E4A7 :
STRUCT
	{attribute addProperty Name "ID"}
	ID : ID_07C9D28F;
	{attribute addProperty Name "WcState"}
	WcState : WcState_9091E0EB;
	{attribute addProperty Name "InfoData"}
	InfoData : InfoData_6F19DB2B;
END_STRUCT
END_TYPE

// ---- DUTs/IO/Boxes/EK1561_1FC0878B.TcDUT
{attribute 'GeneratedUsingTerminal: EK1561-0000-0018'}
{attribute addProperty BoxType "EK1561-0000-0018"}
{attribute addProperty Description "EK1561 1 port EtherCAT junction (POF)"}
{attribute addProperty Physics "K_KY"}
{attribute addProperty Id "InfoDataAT %I*InfoData_6F19DB2B2"}
{attribute addProperty CRC "532711307"}
{attribute addProperty Size "2"}
TYPE EK1561_1FC0878B EXTENDS EtcSlaveTerminalBase_947E5A46 :
STRUCT
	{attribute addProperty Name "InfoData"}
	InfoData : InfoData_6F19DB2B;
END_STRUCT
END_TYPE

// ---- DUTs/IO/Boxes/EK1521_1FC0878B.TcDUT
{attribute 'GeneratedUsingTerminal: EK1521-0010-0020'}
{attribute addProperty BoxType "EK1521-0010-0020"}
{attribute addProperty Description "EK1521-0010 1 port EtherCAT junction (FX-SingleMode)"}
{attribute addProperty Physics "K_KY"}
{attribute addProperty Id "InfoDataAT %I*InfoData_6F19DB2B2"}
{attribute addProperty CRC "532711307"}
{attribute addProperty Size "2"}
TYPE EK1521_1FC0878B EXTENDS EtcSlaveTerminalBase_947E5A46 :
STRUCT
	{attribute addProperty Name "InfoData"}
	InfoData : InfoData_6F19DB2B;
END_STRUCT
END_TYPE

// ---- DUTs/IO/Boxes/EK1814_F6D9A8D1.TcDUT
{attribute 'GeneratedUsingTerminal: EK1814-0000-0016'}
{attribute addProperty BoxType "EK1814-0000-0016"}
{attribute addProperty Description "EK1814 EtherCAT IO-Coupler  (0,5A E-Bus, 4 Ch. Dig. In, 3ms, 4 Ch. Dig. Out 24V, 0,5A)"}
{attribute addProperty Physics "YKY"}
{attribute addProperty Id "Channel_1AT %I*Channel_830843C11Channel_2AT %I*Channel_830843C11Channel_3AT %I*Channel_830843C11Channel_4AT %I*Channel_830843C11Channel_5AT %Q*Channel_42CA91F71Channel_6AT %Q*Channel_42CA91F71Channel_7AT %Q*Channel_42CA91F71Channel_8AT %Q*Channel_42CA91F71WcStateAT %I*WcState_9091E0EB2InfoDataAT %I*InfoData_6F19DB2B2"}
{attribute addProperty CRC "4141459665"}
{attribute addProperty Size "12"}
TYPE EK1814_F6D9A8D1 EXTENDS EtcSlaveBoxBase_77A0E4A7 :
STRUCT
	{attribute addProperty Name "Channel_1"}
	Channel_1 : Channel_830843C1;
	{attribute addProperty Name "Channel_2"}
	Channel_2 : Channel_830843C1;
	{attribute addProperty Name "Channel_3"}
	Channel_3 : Channel_830843C1;
	{attribute addProperty Name "Channel_4"}
	Channel_4 : Channel_830843C1;
	{attribute addProperty Name "Channel_5"}
	Channel_5 : Channel_42CA91F7;
	{attribute addProperty Name "Channel_6"}
	Channel_6 : Channel_42CA91F7;
	{attribute addProperty Name "Channel_7"}
	Channel_7 : Channel_42CA91F7;
	{attribute addProperty Name "Channel_8"}
	Channel_8 : Channel_42CA91F7;
	{attribute addProperty Name "WcState"}
	WcState : WcState_9091E0EB;
	{attribute addProperty Name "InfoData"}
	InfoData : InfoData_6F19DB2B;
END_STRUCT
END_TYPE

// ---- DUTs/IO/Boxes/EK1818_6B19C24E.TcDUT
{attribute 'GeneratedUsingTerminal: EK1818-0000-0016'}
{attribute addProperty BoxType "EK1818-0000-0016"}
{attribute addProperty Description "EK1818 EtherCAT IO-Coupler  (1A E-Bus, 8 Ch. Dig. In, 3ms, 4 Ch. Dig. Out 24V, 0,5A)"}
{attribute addProperty Physics "YKY"}
{attribute addProperty Id "Channel_1AT %I*Channel_830843C11Channel_2AT %I*Channel_830843C11Channel_3AT %I*Channel_830843C11Channel_4AT %I*Channel_830843C11Channel_5AT %I*Channel_830843C11Channel_6AT %I*Channel_830843C11Channel_7AT %I*Channel_830843C11Channel_8AT %I*Channel_830843C11Channel_9AT %Q*Channel_42CA91F71Channel_10AT %Q*Channel_42CA91F71Channel_11AT %Q*Channel_42CA91F71Channel_12AT %Q*Channel_42CA91F71WcStateAT %I*WcState_9091E0EB2InfoDataAT %I*InfoData_6F19DB2B2"}
{attribute addProperty CRC "1796850254"}
{attribute addProperty Size "16"}
TYPE EK1818_6B19C24E EXTENDS EtcSlaveBoxBase_77A0E4A7 :
STRUCT
	{attribute addProperty Name "Channel_1"}
	Channel_1 : Channel_830843C1;
	{attribute addProperty Name "Channel_2"}
	Channel_2 : Channel_830843C1;
	{attribute addProperty Name "Channel_3"}
	Channel_3 : Channel_830843C1;
	{attribute addProperty Name "Channel_4"}
	Channel_4 : Channel_830843C1;
	{attribute addProperty Name "Channel_5"}
	Channel_5 : Channel_830843C1;
	{attribute addProperty Name "Channel_6"}
	Channel_6 : Channel_830843C1;
	{attribute addProperty Name "Channel_7"}
	Channel_7 : Channel_830843C1;
	{attribute addProperty Name "Channel_8"}
	Channel_8 : Channel_830843C1;
	{attribute addProperty Name "Channel_9"}
	Channel_9 : Channel_42CA91F7;
	{attribute addProperty Name "Channel_10"}
	Channel_10 : Channel_42CA91F7;
	{attribute addProperty Name "Channel_11"}
	Channel_11 : Channel_42CA91F7;
	{attribute addProperty Name "Channel_12"}
	Channel_12 : Channel_42CA91F7;
	{attribute addProperty Name "WcState"}
	WcState : WcState_9091E0EB;
	{attribute addProperty Name "InfoData"}
	InfoData : InfoData_6F19DB2B;
END_STRUCT
END_TYPE

// ---- DUTs/IO/Boxes/EK1828_56D6F887.TcDUT
{attribute 'GeneratedUsingTerminal: EK1828-0000-0016'}
{attribute addProperty BoxType "EK1828-0000-0016"}
{attribute addProperty Description "EK1828 EtherCAT IO-Coupler  (1A E-Bus, 4 Ch. Dig. In, 3ms, 8 Ch. Dig. Out 24V, 0,5A)"}
{attribute addProperty Physics "YKY"}
{attribute addProperty Id "Channel_1AT %I*Channel_830843C11Channel_2AT %I*Channel_830843C11Channel_3AT %I*Channel_830843C11Channel_4AT %I*Channel_830843C11Channel_5AT %Q*Channel_42CA91F71Channel_6AT %Q*Channel_42CA91F71Channel_7AT %Q*Channel_42CA91F71Channel_8AT %Q*Channel_42CA91F71Channel_9AT %Q*Channel_42CA91F71Channel_10AT %Q*Channel_42CA91F71Channel_11AT %Q*Channel_42CA91F71Channel_12AT %Q*Channel_42CA91F71WcStateAT %I*WcState_9091E0EB2InfoDataAT %I*InfoData_6F19DB2B2"}
{attribute addProperty CRC "1456928903"}
{attribute addProperty Size "16"}
TYPE EK1828_56D6F887 EXTENDS EtcSlaveBoxBase_77A0E4A7 :
STRUCT
	{attribute addProperty Name "Channel_1"}
	Channel_1 : Channel_830843C1;
	{attribute addProperty Name "Channel_2"}
	Channel_2 : Channel_830843C1;
	{attribute addProperty Name "Channel_3"}
	Channel_3 : Channel_830843C1;
	{attribute addProperty Name "Channel_4"}
	Channel_4 : Channel_830843C1;
	{attribute addProperty Name "Channel_5"}
	Channel_5 : Channel_42CA91F7;
	{attribute addProperty Name "Channel_6"}
	Channel_6 : Channel_42CA91F7;
	{attribute addProperty Name "Channel_7"}
	Channel_7 : Channel_42CA91F7;
	{attribute addProperty Name "Channel_8"}
	Channel_8 : Channel_42CA91F7;
	{attribute addProperty Name "Channel_9"}
	Channel_9 : Channel_42CA91F7;
	{attribute addProperty Name "Channel_10"}
	Channel_10 : Channel_42CA91F7;
	{attribute addProperty Name "Channel_11"}
	Channel_11 : Channel_42CA91F7;
	{attribute addProperty Name "Channel_12"}
	Channel_12 : Channel_42CA91F7;
	{attribute addProperty Name "WcState"}
	WcState : WcState_9091E0EB;
	{attribute addProperty Name "InfoData"}
	InfoData : InfoData_6F19DB2B;
END_STRUCT
END_TYPE

// ---- DUTs/IO/Boxes/EK1828_E2806B95.TcDUT
{attribute 'GeneratedUsingTerminal: EK1828-0010-0016'}
{attribute addProperty BoxType "EK1828-0010-0016"}
{attribute addProperty Description "EK1828-0010 EtherCAT IO-Coupler  (1A E-Bus, 8 Ch. Dig. Out 24V, 0,5A)"}
{attribute addProperty Physics "YKY"}
{attribute addProperty Id "Channel_1AT %Q*Channel_42CA91F71Channel_2AT %Q*Channel_42CA91F71Channel_3AT %Q*Channel_42CA91F71Channel_4AT %Q*Channel_42CA91F71Channel_5AT %Q*Channel_42CA91F71Channel_6AT %Q*Channel_42CA91F71Channel_7AT %Q*Channel_42CA91F71Channel_8AT %Q*Channel_42CA91F71WcStateAT %I*WcState_0B2B16F91InfoDataAT %I*InfoData_6F19DB2B2"}
{attribute addProperty CRC "3800066965"}
{attribute addProperty Size "11"}
TYPE EK1828_E2806B95 EXTENDS EtcSlaveBoxBase_77A0E4A7 :
STRUCT
	{attribute addProperty Name "Channel_1"}
	Channel_1 : Channel_42CA91F7;
	{attribute addProperty Name "Channel_2"}
	Channel_2 : Channel_42CA91F7;
	{attribute addProperty Name "Channel_3"}
	Channel_3 : Channel_42CA91F7;
	{attribute addProperty Name "Channel_4"}
	Channel_4 : Channel_42CA91F7;
	{attribute addProperty Name "Channel_5"}
	Channel_5 : Channel_42CA91F7;
	{attribute addProperty Name "Channel_6"}
	Channel_6 : Channel_42CA91F7;
	{attribute addProperty Name "Channel_7"}
	Channel_7 : Channel_42CA91F7;
	{attribute addProperty Name "Channel_8"}
	Channel_8 : Channel_42CA91F7;
	{attribute addProperty Name "WcState"}
	WcState : WcState_0B2B16F9;
	{attribute addProperty Name "InfoData"}
	InfoData : InfoData_6F19DB2B;
END_STRUCT
END_TYPE

// ---- DUTs/IO/Boxes/EKM1101_7F417622.TcDUT
{attribute 'GeneratedUsingTerminal: EKM1101-0000-0016'}
{attribute addProperty BoxType "EKM1101-0000-0016"}
{attribute addProperty Description "EKM1101 EtherCAT Coupler  (2A E-Bus, ID switch, Diagnostics, isolated)"}
{attribute addProperty Physics "YKY"}
{attribute addProperty Id "MMS_Device_InputsAT %I*MMS_Device_Inputs_ADC3123E5MMS_Acceleration_StatusAT %I*MMS_Acceleration_Status_117690999MMS_Acceleration_X_AxisAT %I*MMS_Acceleration_X_Axis_80E77D6A2MMS_Acceleration_Y_AxisAT %I*MMS_Acceleration_Y_Axis_80E77D6A2MMS_Acceleration_Z_AxisAT %I*MMS_Acceleration_Z_Axis_80E77D6A2MMS_Acceleration_TimestampAT %I*MMS_Acceleration_Timestamp_8B9FE1A28MMS_Voltage_Us_In_InputsAT %I*MMS_Voltage_Us_In_Inputs_60D55C7211MMS_Voltage_Up_In_InputsAT %I*MMS_Voltage_Up_In_Inputs_60D55C7211MMS_Voltage_Up_Out_InputsAT %I*MMS_Voltage_Up_Out_Inputs_60D55C7211MMS_Device_OutputsAT %Q*MMS_Device_Outputs_E6E6F9D11WcStateAT %I*WcState_9091E0EB2InfoDataAT %I*InfoData_BEF6B88E18"}
{attribute addProperty CRC "2134996514"}
{attribute addProperty Size "82"}
TYPE EKM1101_7F417622 EXTENDS EtcSlaveBoxBase_77A0E4A7 :
STRUCT
	{attribute addProperty Name "MMS_Device_Inputs"}
	MMS_Device_Inputs : MMS_Device_Inputs_ADC3123E;
	{attribute addProperty Name "MMS_Acceleration_Status"}
	MMS_Acceleration_Status : MMS_Acceleration_Status_11769099;
	{attribute addProperty Name "MMS_Acceleration_X_Axis"}
	MMS_Acceleration_X_Axis : MMS_Acceleration_X_Axis_80E77D6A;
	{attribute addProperty Name "MMS_Acceleration_Y_Axis"}
	MMS_Acceleration_Y_Axis : MMS_Acceleration_Y_Axis_80E77D6A;
	{attribute addProperty Name "MMS_Acceleration_Z_Axis"}
	MMS_Acceleration_Z_Axis : MMS_Acceleration_Z_Axis_80E77D6A;
	{attribute addProperty Name "MMS_Acceleration_Timestamp"}
	MMS_Acceleration_Timestamp : MMS_Acceleration_Timestamp_8B9FE1A2;
	{attribute addProperty Name "MMS_Voltage_Us_In_Inputs"}
	MMS_Voltage_Us_In_Inputs : MMS_Voltage_Us_In_Inputs_60D55C72;
	{attribute addProperty Name "MMS_Voltage_Up_In_Inputs"}
	MMS_Voltage_Up_In_Inputs : MMS_Voltage_Up_In_Inputs_60D55C72;
	{attribute addProperty Name "MMS_Voltage_Up_Out_Inputs"}
	MMS_Voltage_Up_Out_Inputs : MMS_Voltage_Up_Out_Inputs_60D55C72;
	{attribute addProperty Name "MMS_Device_Outputs"}
	MMS_Device_Outputs : MMS_Device_Outputs_E6E6F9D1;
	{attribute addProperty Name "WcState"}
	WcState : WcState_9091E0EB;
	{attribute addProperty Name "InfoData"}
	InfoData : InfoData_BEF6B88E;
END_STRUCT
END_TYPE

// ---- DUTs/IO/Boxes/EK1960_14394C51.TcDUT
{attribute 'GeneratedUsingTerminal: EK1960-0000-0019'}
{attribute addProperty BoxType "EK1960-0000-0019"}
{attribute addProperty Description "EK1960-0000 TwinSAFE-Compact-Controller (RJ45)"}
{attribute addProperty Physics "YKY"}
{attribute addProperty Id "Module_1_FSoEModule_1_FSoE_BE928FF798Module_2_FSOUTModule_2_FSOUT_E84B1B0028Module_3_FSLOGICModule_3_FSLOGIC_DEAB45222WcStateAT %I*WcState_B516A2644InfoDataAT %I*InfoData_32EB74EA10"}
{attribute addProperty CRC "339299409"}
{attribute addProperty Size "142"}
TYPE EK1960_14394C51 EXTENDS EtcSlaveBoxBase_77A0E4A7 :
STRUCT
	{attribute addProperty Name "Module_1_FSoE"}
	Module_1_FSoE : Module_1_FSoE_BE928FF7;
	{attribute addProperty Name "Module_2_FSOUT"}
	Module_2_FSOUT : Module_2_FSOUT_E84B1B00;
	{attribute addProperty Name "Module_3_FSLOGIC"}
	Module_3_FSLOGIC : Module_3_FSLOGIC_DEAB4522;
	{attribute addProperty Name "WcState"}
	WcState : WcState_B516A264;
	{attribute addProperty Name "InfoData"}
	InfoData : InfoData_32EB74EA;
END_STRUCT
END_TYPE

// ---- DUTs/IO/Boxes/EK1960_9900B192.TcDUT
{attribute 'GeneratedUsingTerminal: EK1960-0000-0021'}
{attribute addProperty BoxType "EK1960-0000-0021"}
{attribute addProperty Description "EK1960-0000 TwinSAFE-Compact-Controller (RJ45)"}
{attribute addProperty Physics "YKY"}
{attribute addProperty Id "Module_1_FSoEModule_1_FSoE_042BAFD398Module_2_FSOUTModule_2_FSOUT_8B7AA8A224Module_3_FSLOGICModule_3_FSLOGIC_DEAB45222WcStateAT %I*WcState_B516A2644InfoDataAT %I*InfoData_32EB74EA10"}
{attribute addProperty CRC "2566959506"}
{attribute addProperty Size "138"}
TYPE EK1960_9900B192 EXTENDS EtcSlaveBoxBase_77A0E4A7 :
STRUCT
	{attribute addProperty Name "Module_1_FSoE"}
	Module_1_FSoE : Module_1_FSoE_042BAFD3;
	{attribute addProperty Name "Module_2_FSOUT"}
	Module_2_FSOUT : Module_2_FSOUT_8B7AA8A2;
	{attribute addProperty Name "Module_3_FSLOGIC"}
	Module_3_FSLOGIC : Module_3_FSLOGIC_DEAB4522;
	{attribute addProperty Name "WcState"}
	WcState : WcState_B516A264;
	{attribute addProperty Name "InfoData"}
	InfoData : InfoData_32EB74EA;
END_STRUCT
END_TYPE

// ---- DUTs/IO/Boxes/EK1960_BAE25DEC.TcDUT
{attribute 'GeneratedUsingTerminal: EK1960-2600-0019'}
{attribute addProperty BoxType "EK1960-2600-0019"}
{attribute addProperty Description "EK1960-2600 TwinSAFE-Compact-Controller (4 x Relay, RJ45)"}
{attribute addProperty Physics "YKY"}
{attribute addProperty Id "Module_1_FSoEModule_1_FSoE_7E6C60DE104Module_2_FSOUTModule_2_FSOUT_E84B1B0028Module_3_FSLOGICModule_3_FSLOGIC_DEAB45222WcStateAT %I*WcState_B516A2644InfoDataAT %I*InfoData_32EB74EA10"}
{attribute addProperty CRC "3135397356"}
{attribute addProperty Size "148"}
TYPE EK1960_BAE25DEC EXTENDS EtcSlaveBoxBase_77A0E4A7 :
STRUCT
	{attribute addProperty Name "Module_1_FSoE"}
	Module_1_FSoE : Module_1_FSoE_7E6C60DE;
	{attribute addProperty Name "Module_2_FSOUT"}
	Module_2_FSOUT : Module_2_FSOUT_E84B1B00;
	{attribute addProperty Name "Module_3_FSLOGIC"}
	Module_3_FSLOGIC : Module_3_FSLOGIC_DEAB4522;
	{attribute addProperty Name "WcState"}
	WcState : WcState_B516A264;
	{attribute addProperty Name "InfoData"}
	InfoData : InfoData_32EB74EA;
END_STRUCT
END_TYPE

// ---- DUTs/IO/Boxes/EK1960_2415CDAE.TcDUT
{attribute 'GeneratedUsingTerminal: EK1960-2600-0021'}
{attribute addProperty BoxType "EK1960-2600-0021"}
{attribute addProperty Description "EK1960-2600 TwinSAFE-Compact-Controller (4 x Relay, RJ45)"}
{attribute addProperty Physics "YKY"}
{attribute addProperty Id "Module_1_FSoEModule_1_FSoE_B78AD590104Module_2_FSOUTModule_2_FSOUT_E84B1B0028Module_3_FSLOGICModule_3_FSLOGIC_DEAB45222WcStateAT %I*WcState_B516A2644InfoDataAT %I*InfoData_32EB74EA10"}
{attribute addProperty CRC "605408686"}
{attribute addProperty Size "148"}
TYPE EK1960_2415CDAE EXTENDS EtcSlaveBoxBase_77A0E4A7 :
STRUCT
	{attribute addProperty Name "Module_1_FSoE"}
	Module_1_FSoE : Module_1_FSoE_B78AD590;
	{attribute addProperty Name "Module_2_FSOUT"}
	Module_2_FSOUT : Module_2_FSOUT_E84B1B00;
	{attribute addProperty Name "Module_3_FSLOGIC"}
	Module_3_FSLOGIC : Module_3_FSLOGIC_DEAB4522;
	{attribute addProperty Name "WcState"}
	WcState : WcState_B516A264;
	{attribute addProperty Name "InfoData"}
	InfoData : InfoData_32EB74EA;
END_STRUCT
END_TYPE

// ---- DUTs/IO/Devices/SyncUnitTask_2D604ED5.TcDUT
{attribute 'GeneratedUsingTerminal: IODEVICETYPE_ETHERCATPROT'}
{attribute addProperty BoxType "IODEVICETYPE_ETHERCATPROT"}
{attribute addProperty Id "WcStateAT %I*WcState_0B2B16F91InfoDataAT %I*InfoData_2A97D6CF8"}
{attribute addProperty CRC "761286357"}
{attribute addProperty Size "9"}
TYPE SyncUnitTask_2D604ED5 :
STRUCT
	{attribute addProperty Name "WcState"}
	WcState : WcState_0B2B16F9;
	{attribute addProperty Name "InfoData"}
	InfoData : InfoData_2A97D6CF;
END_STRUCT
END_TYPE

// ---- DUTs/IO/Devices/SyncUnitTasks_6FEB8257.TcDUT
{attribute 'GeneratedUsingTerminal: '}
{attribute addProperty BoxType ""}
{attribute addProperty Id "unreferencedAT %I*SyncUnitTask_2D604ED59PlcTaskAT %I*SyncUnitTask_2D604ED59"}
{attribute addProperty CRC "1877705303"}
{attribute addProperty Size "18"}
TYPE SyncUnitTasks_6FEB8257 :
STRUCT
	{attribute addProperty Name "unreferenced"}
	unreferenced : SyncUnitTask_2D604ED5;
	{attribute addProperty Name "PlcTask"}
	PlcTask : SyncUnitTask_2D604ED5;
END_STRUCT
END_TYPE

// ---- DUTs/IO/Devices/SyncUnits_99E584AF.TcDUT
{attribute 'GeneratedUsingTerminal: '}
{attribute addProperty BoxType ""}
{attribute addProperty Id "_defaultAT %I*SyncUnitTasks_6FEB825718"}
{attribute addProperty CRC "2581955759"}
{attribute addProperty Size "18"}
TYPE SyncUnits_99E584AF :
STRUCT
	{attribute addProperty Name "_default"}
	_default : SyncUnitTasks_6FEB8257;
END_STRUCT
END_TYPE

// ---- DUTs/IO/Topology/Beckhoff_EK11xxEK1122_42F1D1D1.TcDUT
{attribute 'GeneratedUsingTerminal: EK1122-0000-0018'}
{attribute addProperty BoxType "EK1122-0000-0018"}
{attribute addProperty Id "Beckhoff_EK11xxsub_EK1100EK1100_1FC0878B2A_0001_EK1100_0000_0000EK1100_1FC0878B2A_0002_EK1100_0000_0001EK1100_1FC0878B2A_0003_EK1100_0000_0016EK1100_1FC0878B2A_0004_EK1100_0000_0017EK1100_1FC0878B2A_0005_EK1100_0000_0018EK1100_1FC0878B2A_0006_EK1100_0008_0016EK1100_1FC0878B2A_0009_EK1101_0000_0016EK1101_957D888F6A_0010_EK1101_0000_0017EK1101_957D888F6A_0011_EK1101_0000_0018EK1101_957D888F6A_0012_EK1101_0008_0016EK1101_957D888F6A_0013_EK1101_0010_0016EK1101_957D888F6A_0008_EK1100_0030_0017EK1100_1FC0878B2A_0007_EK1100_0030_0016EK1100_1FC0878B2"}
{attribute addProperty CRC "1123144145"}
{attribute addProperty Size "48"}
{attribute addProperty Name "Beckhoff EK11xxEK1122"}
TYPE Beckhoff_EK11xxEK1122_42F1D1D1 EXTENDS EK1122_1FC0878B :
STRUCT
	{attribute addProperty Name "Beckhoff EK11xxsub EK1100"}
	{attribute addProperty PreviousPort "Beckhoff EK11xxEK1122 : D"}
	Beckhoff_EK11xxsub_EK1100 : EK1100_1FC0878B;
	{attribute addProperty Name "A_0001(EK1100-0000-0000)"}
	{attribute addProperty PreviousPort "Beckhoff EK11xxsub EK1100 : C"}
	A_0001_EK1100_0000_0000 : EK1100_1FC0878B;
	{attribute addProperty Name "A_0002(EK1100-0000-0001)"}
	{attribute addProperty PreviousPort "A_0001(EK1100-0000-0000) : C"}
	A_0002_EK1100_0000_0001 : EK1100_1FC0878B;
	{attribute addProperty Name "A_0003(EK1100-0000-0016)"}
	{attribute addProperty PreviousPort "A_0002(EK1100-0000-0001) : C"}
	A_0003_EK1100_0000_0016 : EK1100_1FC0878B;
	{attribute addProperty Name "A_0004(EK1100-0000-0017)"}
	{attribute addProperty PreviousPort "A_0003(EK1100-0000-0016) : C"}
	A_0004_EK1100_0000_0017 : EK1100_1FC0878B;
	{attribute addProperty Name "A_0005(EK1100-0000-0018)"}
	{attribute addProperty PreviousPort "A_0004(EK1100-0000-0017) : C"}
	A_0005_EK1100_0000_0018 : EK1100_1FC0878B;
	{attribute addProperty Name "A_0006(EK1100-0008-0016)"}
	{attribute addProperty PreviousPort "A_0005(EK1100-0000-0018) : C"}
	A_0006_EK1100_0008_0016 : EK1100_1FC0878B;
	{attribute addProperty Name "A_0009(EK1101-0000-0016)"}
	{attribute addProperty PreviousPort "A_0006(EK1100-0008-0016) : C"}
	A_0009_EK1101_0000_0016 : EK1101_957D888F;
	{attribute addProperty Name "A_0010(EK1101-0000-0017)"}
	{attribute addProperty PreviousPort "A_0009(EK1101-0000-0016) : C"}
	A_0010_EK1101_0000_0017 : EK1101_957D888F;
	{attribute addProperty Name "A_0011(EK1101-0000-0018)"}
	{attribute addProperty PreviousPort "A_0010(EK1101-0000-0017) : C"}
	A_0011_EK1101_0000_0018 : EK1101_957D888F;
	{attribute addProperty Name "A_0012(EK1101-0008-0016)"}
	{attribute addProperty PreviousPort "A_0011(EK1101-0000-0018) : C"}
	A_0012_EK1101_0008_0016 : EK1101_957D888F;
	{attribute addProperty Name "A_0013(EK1101-0010-0016)"}
	{attribute addProperty PreviousPort "A_0012(EK1101-0008-0016) : C"}
	A_0013_EK1101_0010_0016 : EK1101_957D888F;
	{attribute addProperty Name "A_0008(EK1100-0030-0017)"}
	{attribute addProperty PreviousPort "A_0013(EK1101-0010-0016) : C"}
	A_0008_EK1100_0030_0017 : EK1100_1FC0878B;
	{attribute addProperty Name "A_0007(EK1100-0030-0016)"}
	{attribute addProperty PreviousPort "Beckhoff EK11xxEK1122 : B"}
	A_0007_EK1100_0030_0016 : EK1100_1FC0878B;
END_STRUCT
END_TYPE

// ---- DUTs/IO/Topology/Beckhoff_EK11xx_811529C6.TcDUT
{attribute 'GeneratedUsingTerminal: EK1100-0000-0018'}
{attribute addProperty BoxType "EK1100-0000-0018"}
{attribute addProperty Id "Beckhoff_EK11xxEK1122Beckhoff_EK11xxEK1122_42F1D1D148A_0018_EK1110_0043_0016EK1110_1FC0878B2A_0024_EK1122_0008_0016EK1122_1FC0878B2A_0023_EK1122_0000_0018EK1122_1FC0878B2A_0022_EK1122_0000_0017EK1122_1FC0878B2A_0021_EK1122_0000_0016EK1122_1FC0878B2A_0020_EK1121_0010_0016EK1121_1FC0878B2A_0019_EK1110_0044_0016EK1110_1FC0878B2A_0017_EK1110_0008_0016EK1110_1FC0878B2A_0016_EK1110_0000_0017EK1110_1FC0878B2A_0015_EK1110_0000_0016EK1110_1FC0878B2A_0014_EK1110_0000_0000EK1110_1FC0878B2"}
{attribute addProperty CRC "2165647814"}
{attribute addProperty Size "70"}
{attribute addProperty Name "Beckhoff EK11xx"}
TYPE Beckhoff_EK11xx_811529C6 EXTENDS EK1100_1FC0878B :
STRUCT
	{attribute addProperty Name "Beckhoff EK11xxEK1122"}
	{attribute addProperty PreviousPort "Beckhoff EK11xx : B"}
	Beckhoff_EK11xxEK1122 : Beckhoff_EK11xxEK1122_42F1D1D1;
	{attribute addProperty Name "A_0018(EK1110-0043-0016)"}
	{attribute addProperty PreviousPort "Beckhoff EK11xxEK1122 : C"}
	A_0018_EK1110_0043_0016 : EK1110_1FC0878B;
	{attribute addProperty Name "A_0024(EK1122-0008-0016)"}
	{attribute addProperty PreviousPort "A_0018(EK1110-0043-0016) : B"}
	A_0024_EK1122_0008_0016 : EK1122_1FC0878B;
	{attribute addProperty Name "A_0023(EK1122-0000-0018)"}
	{attribute addProperty PreviousPort "A_0024(EK1122-0008-0016) : C"}
	A_0023_EK1122_0000_0018 : EK1122_1FC0878B;
	{attribute addProperty Name "A_0022(EK1122-0000-0017)"}
	{attribute addProperty PreviousPort "A_0023(EK1122-0000-0018) : C"}
	A_0022_EK1122_0000_0017 : EK1122_1FC0878B;
	{attribute addProperty Name "A_0021(EK1122-0000-0016)"}
	{attribute addProperty PreviousPort "A_0022(EK1122-0000-0017) : C"}
	A_0021_EK1122_0000_0016 : EK1122_1FC0878B;
	{attribute addProperty Name "A_0020(EK1121-0010-0016)"}
	{attribute addProperty PreviousPort "A_0021(EK1122-0000-0016) : C"}
	A_0020_EK1121_0010_0016 : EK1121_1FC0878B;
	{attribute addProperty Name "A_0019(EK1110-0044-0016)"}
	{attribute addProperty PreviousPort "A_0020(EK1121-0010-0016) : C"}
	A_0019_EK1110_0044_0016 : EK1110_1FC0878B;
	{attribute addProperty Name "A_0017(EK1110-0008-0016)"}
	{attribute addProperty PreviousPort "A_0019(EK1110-0044-0016) : B"}
	A_0017_EK1110_0008_0016 : EK1110_1FC0878B;
	{attribute addProperty Name "A_0016(EK1110-0000-0017)"}
	{attribute addProperty PreviousPort "Beckhoff EK11xxEK1122 : C"}
	A_0016_EK1110_0000_0017 : EK1110_1FC0878B;
	{attribute addProperty Name "A_0015(EK1110-0000-0016)"}
	{attribute addProperty PreviousPort "Beckhoff EK11xxEK1122 : C"}
	A_0015_EK1110_0000_0016 : EK1110_1FC0878B;
	{attribute addProperty Name "A_0014(EK1110-0000-0000)"}
	{attribute addProperty PreviousPort "Beckhoff EK11xxEK1122 : C"}
	A_0014_EK1110_0000_0000 : EK1110_1FC0878B;
END_STRUCT
END_TYPE

